KUKA KRL program: EPS_2_25694_HR02_A_20260114065909.src

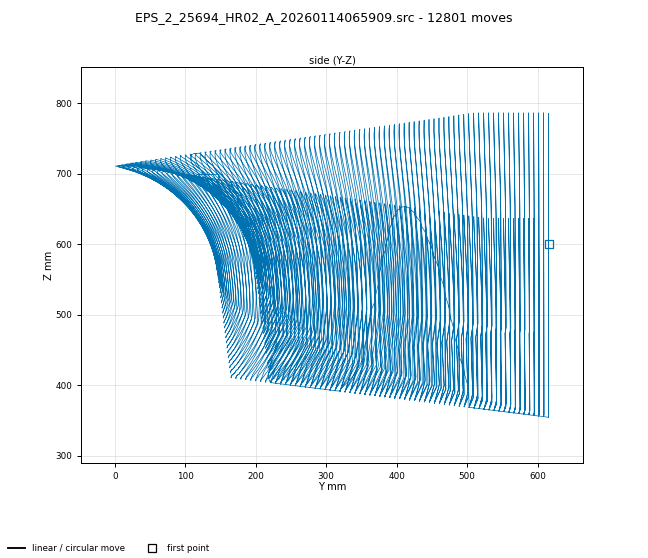
[picture p0: tool path of EPS_2_25694_HR02_A_20260114065909.src, 12801 of 12803 moves have a stored position in this frame; points joined in program order, loops and branches not executed]
&ACCESS RVP
&REL 4
&COMMENT QRS 19112012
&PARAM EDITMASK = *
DEF PART()
EXT BAS (BAS_COMMAND :IN,REAL :IN )
INT I
BAS (#INITMOV,0 )

;KUKA QRS Post kuka4.cps  Date:22-06-2017 !

File_ID=2967

QRS_PRE_INIT()

;Init var - Until changes are made in qrs_pre_init
Outlet_Square_prg=0
Inlet_1_Square_prg=0
Inlet_2_Square_prg=0
Inlet_3_Square_prg=0
Inlet_4_Square_prg=0
Inlet_5_Square_prg=0

Outlet_1={X 0.000, Y 512.360, Z 637.000, B 0.000, E1 0.000 }
Inlet_1={X 0.000, Y 526.980, Z 437.000, B 0.000, E1 171.000 }
Outlet_1_type=299
Inlet_1_type=299
;QRS#1=Sidecore dimensions
;QRS#2=300-12" PVC SDR 35
;QRS#3=300-12" PVC SDR 35
;QRS#4=
;QRS#5=
;QRS#6=
;QRS#7=
;QRS#8=
;QRS#9=16M PSX
;QRS#10=16M PSX
;QRS#11=
;QRS#12=
;QRS#13=
;QRS#14=
;QRS#15=
;QRS#16=1220x127x1067 3,5'
;QRS#17=EPS Height
;QRS#18=786,5
;QRS#19=*
;QRS#20= UPDATED VERSION 22-06-2017
;QRS#21=*
Outlet_Square=0150
Inlet_1_Square=0150
Inlet_2_Square=0
Inlet_3_Square=0
Inlet_4_Square=0
Inlet_5_Square=0
Mill_Square=1
Outlet_Square_Prg=206
Inlet_1_Square_prg=206

QRS_INIT()

$ADVANCE=5

; T1
PTP {E1 173.595,E2 173.595}
PTP {X 0,Y 615.516,A -85,B 0,C 180,E1 173.595,E2 173.595,E3 0,E4 0,E5 0,E6 0}
QRS_SPEED_INIT()
LIN {X 0,Y 615.516,Z 600,A -85,B 0,C 180,E1 173.595,E2 173.595,E3 0,E4 0,E5 0,E6 0} C_VEL
LIN {X 0,Y 615.516,Z 364.494,A -85,B 0,C 180,E1 173.595,E2 173.595} C_VEL
LIN {X 0,Y 615.516,Z 356.327,A -85,B 0,C 180,E1 173.595,E2 173.595} C_VEL
LIN {X 0,Y 615.485,Z 354.327,A -85,B 0,C 180,E1 173.409,E2 173.409} C_VEL
LIN {X 0,Y 615.431,Z 354.324,A -85,B 0,C 180,E1 170.8,E2 170.8} C_VEL
LIN {X 0,Y 615.434,Z 354.324,A -85,B 0,C 180,E1 168.806,E2 168.806} C_VEL
LIN {X 0,Y 615.435,Z 354.324,A -85,B 0,C 180,E1 166.797,E2 166.797} C_VEL
LIN {X 0,Y 615.435,Z 354.324,A -85,B 0,C 180,E1 164.772,E2 164.772} C_VEL
LIN {X 0,Y 615.433,Z 354.323,A -85,B 0,C 180,E1 162.728,E2 162.728} C_VEL
LIN {X 0,Y 615.43,Z 354.323,A -85,B 0,C 180,E1 160.66,E2 160.66} C_VEL
LIN {X 0,Y 615.426,Z 354.323,A -85,B 0,C 180,E1 158.566,E2 158.566} C_VEL
LIN {X 0,Y 615.422,Z 354.322,A -85,B 0,C 180,E1 156.441,E2 156.441} C_VEL
LIN {X 0,Y 615.421,Z 354.322,A -85,B 0,C 180,E1 154.281,E2 154.281} C_VEL
LIN {X 0,Y 615.468,Z 354.319,A -85,B 0,C 180,E1 151.55,E2 151.55} C_VEL
LIN {X 0,Y 615.466,Z 354.324,A -85,B 0,C 180,E1 148.914,E2 148.914} C_VEL
LIN {X 0,Y 615.43,Z 354.322,A -85,B 0,C 180,E1 146.471,E2 146.471} C_VEL
LIN {X 0,Y 615.424,Z 354.321,A -85,B 0,C 180,E1 144.172,E2 144.172} C_VEL
LIN {X 0,Y 615.431,Z 354.32,A -85,B 0,C 180,E1 141.927,E2 141.927} C_VEL
LIN {X 0,Y 615.474,Z 354.319,A -85,B 0,C 180,E1 139.392,E2 139.392} C_VEL
LIN {X 0,Y 615.462,Z 354.324,A -85,B 0,C 180,E1 136.753,E2 136.753} C_VEL
LIN {X 0,Y 615.484,Z 354.326,A -85,B 0,C 180,E1 134.931,E2 134.931} C_VEL
LIN {X 0,Y 615.433,Z 354.322,A -85,B 0,C 180,E1 132.356,E2 132.356} C_VEL
LIN {X 0,Y 615.427,Z 354.32,A -85,B 0,C 180,E1 130.082,E2 130.082} C_VEL
LIN {X 0,Y 615.429,Z 354.32,A -85,B 0,C 180,E1 128.005,E2 128.005} C_VEL
LIN {X 0,Y 615.444,Z 354.318,A -85,B 0,C 180,E1 125.617,E2 125.617} C_VEL
LIN {X 0,Y 615.481,Z 354.318,A -85,B 0,C 180,E1 123.235,E2 123.235} C_VEL
LIN {X 0,Y 615.494,Z 354.325,A -85,B 0,C 180,E1 120.918,E2 120.918} C_VEL
LIN {X 0,Y 615.45,Z 354.322,A -85,B 0,C 180,E1 118.443,E2 118.443} C_VEL
LIN {X 0,Y 615.491,Z 354.505,A -85,B 0,C 180,E1 116.839,E2 116.839} C_VEL
LIN {X 0,Y 615.483,Z 491.228,A -85,B 0,C 180,E1 115.186,E2 115.186} C_VEL
LIN {X 0,Y 615.499,Z 506.898,A -85,B 0,C 180,E1 114.855,E2 114.855} C_VEL
LIN {X 0,Y 615.488,Z 521.69,A -85,B 0,C 180,E1 114.406,E2 114.406} C_VEL
LIN {X 0,Y 615.489,Z 537.106,A -85,B 0,C 180,E1 113.782,E2 113.782} C_VEL
LIN {X 0,Y 615.497,Z 550.263,A -85,B 0,C 180,E1 113.11,E2 113.11} C_VEL
LIN {X 0,Y 615.497,Z 564.134,A -85,B 0,C 180,E1 112.241,E2 112.241} C_VEL
LIN {X 0,Y 615.498,Z 575.987,A -85,B 0,C 180,E1 111.343,E2 111.343} C_VEL
LIN {X 0,Y 615.496,Z 587.548,A -85,B 0,C 180,E1 110.295,E2 110.295} C_VEL
LIN {X 0,Y 615.497,Z 597.952,A -85,B 0,C 180,E1 109.164,E2 109.164} C_VEL
LIN {X 0,Y 615.497,Z 607.204,A -85,B 0,C 180,E1 107.956,E2 107.956} C_VEL
LIN {X 0,Y 615.493,Z 613.803,A -85,B 0,C 180,E1 106.927,E2 106.927} C_VEL
LIN {X 0,Y 615.496,Z 619.357,A -85,B 0,C 180,E1 105.904,E2 105.904} C_VEL
LIN {X 0,Y 615.493,Z 625.35,A -85,B 0,C 180,E1 104.548,E2 104.548} C_VEL
LIN {X 0,Y 615.493,Z 629.892,A -85,B 0,C 180,E1 103.2,E2 103.2} C_VEL
LIN {X 0,Y 615.49,Z 633.115,A -85,B 0,C 180,E1 101.86,E2 101.86} C_VEL
LIN {X 0,Y 615.489,Z 635.059,A -85,B 0,C 180,E1 100.526,E2 100.526} C_VEL
LIN {X 0,Y 615.49,Z 635.837,A -85,B 0,C 180,E1 99.198,E2 99.198} C_VEL
LIN {X 0,Y 615.497,Z 635.466,A -85,B 0,C 180,E1 97.875,E2 97.875} C_VEL
LIN {X 0,Y 615.495,Z 633.965,A -85,B 0,C 180,E1 96.556,E2 96.556} C_VEL
LIN {X 0,Y 615.495,Z 631.316,A -85,B 0,C 180,E1 95.241,E2 95.241} C_VEL
LIN {X 0,Y 615.491,Z 627.446,A -85,B 0,C 180,E1 93.928,E2 93.928} C_VEL
LIN {X 0,Y 615.488,Z 622.26,A -85,B 0,C 180,E1 92.618,E2 92.618} C_VEL
LIN {X 0,Y 615.49,Z 615.673,A -85,B 0,C 180,E1 91.308,E2 91.308} C_VEL
LIN {X 0,Y 615.497,Z 608.611,A -85,B 0,C 180,E1 90.163,E2 90.163} C_VEL
LIN {X 0,Y 615.494,Z 600.168,A -85,B 0,C 180,E1 89.018,E2 89.018} C_VEL
LIN {X 0,Y 615.495,Z 590.053,A -85,B 0,C 180,E1 87.873,E2 87.873} C_VEL
LIN {X 0,Y 615.497,Z 579.74,A -85,B 0,C 180,E1 86.891,E2 86.891} C_VEL
LIN {X 0,Y 615.499,Z 567.432,A -85,B 0,C 180,E1 85.907,E2 85.907} C_VEL
LIN {X 0,Y 615.498,Z 555.113,A -85,B 0,C 180,E1 85.087,E2 85.087} C_VEL
LIN {X 0,Y 615.482,Z 541.656,A -85,B 0,C 180,E1 84.348,E2 84.348} C_VEL
LIN {X 0,Y 615.485,Z 527.73,A -85,B 0,C 180,E1 83.731,E2 83.731} C_VEL
LIN {X 0,Y 615.49,Z 513.077,A -85,B 0,C 180,E1 83.228,E2 83.228} C_VEL
LIN {X 0,Y 615.481,Z 497.717,A -85,B 0,C 180,E1 82.845,E2 82.845} C_VEL
LIN {X 0,Y 615.449,Z 482.279,A -85,B 0,C 180,E1 82.598,E2 82.598} C_VEL
LIN {X 0,Y 615.499,Z 354.424,A -85,B 0,C 180,E1 81.071,E2 81.071} C_VEL
LIN {X 0,Y 615.479,Z 354.321,A -85,B 0,C 180,E1 78.807,E2 78.807} C_VEL
LIN {X 0,Y 615.417,Z 354.323,A -85,B 0,C 180,E1 76.095,E2 76.095} C_VEL
LIN {X 0,Y 615.417,Z 354.323,A -85,B 0,C 180,E1 74.093,E2 74.093} C_VEL
LIN {X 0,Y 615.416,Z 354.323,A -85,B 0,C 180,E1 72.041,E2 72.041} C_VEL
LIN {X 0,Y 615.436,Z 354.324,A -85,B 0,C 180,E1 69.457,E2 69.457} C_VEL
LIN {X 0,Y 615.441,Z 354.322,A -85,B 0,C 180,E1 66.442,E2 66.442} C_VEL
LIN {X 0,Y 615.428,Z 354.323,A -85,B 0,C 180,E1 64.282,E2 64.282} C_VEL
LIN {X 0,Y 615.417,Z 354.323,A -85,B 0,C 180,E1 62.082,E2 62.082} C_VEL
LIN {X 0,Y 615.413,Z 354.323,A -85,B 0,C 180,E1 59.836,E2 59.836} C_VEL
LIN {X 0,Y 615.422,Z 354.324,A -85,B 0,C 180,E1 57.539,E2 57.539} C_VEL
LIN {X 0,Y 615.453,Z 354.325,A -85,B 0,C 180,E1 55.183,E2 55.183} C_VEL
LIN {X 0,Y 615.488,Z 354.324,A -85,B 0,C 180,E1 52.759,E2 52.759} C_VEL
LIN {X 0,Y 615.43,Z 354.323,A -85,B 0,C 180,E1 50.246,E2 50.246} C_VEL
LIN {X 0,Y 615.413,Z 354.324,A -85,B 0,C 180,E1 47.928,E2 47.928} C_VEL
LIN {X 0,Y 615.41,Z 354.324,A -85,B 0,C 180,E1 45.845,E2 45.845} C_VEL
LIN {X 0,Y 615.435,Z 354.325,A -85,B 0,C 180,E1 43.25,E2 43.25} C_VEL
LIN {X 0,Y 615.467,Z 354.326,A -85,B 0,C 180,E1 40.608,E2 40.608} C_VEL
LIN {X 0,Y 615.417,Z 354.324,A -85,B 0,C 180,E1 38.005,E2 38.005} C_VEL
LIN {X 0,Y 615.41,Z 354.324,A -85,B 0,C 180,E1 35.621,E2 35.621} C_VEL
LIN {X 0,Y 615.429,Z 354.325,A -85,B 0,C 180,E1 33.24,E2 33.24} C_VEL
LIN {X 0,Y 615.46,Z 354.326,A -85,B 0,C 180,E1 30.922,E2 30.922} C_VEL
LIN {X 0,Y 615.464,Z 354.325,A -85,B 0,C 180,E1 28.448,E2 28.448} C_VEL
LIN {X 0,Y 615.408,Z 354.325,A -85,B 0,C 180,E1 25.72,E2 25.72} C_VEL
LIN {X 0,Y 615.408,Z 354.325,A -85,B 0,C 180,E1 23.56,E2 23.56} C_VEL
LIN {X 0,Y 615.41,Z 354.325,A -85,B 0,C 180,E1 21.435,E2 21.435} C_VEL
LIN {X 0,Y 615.48,Z 354.328,A -85,B 0,C 180,E1 18.646,E2 18.646} C_VEL
LIN {X 0,Y 615.416,Z 354.325,A -85,B 0,C 180,E1 15.907,E2 15.907} C_VEL
LIN {X 0,Y 615.415,Z 354.325,A -85,B 0,C 180,E1 13.876,E2 13.876} C_VEL
LIN {X 0,Y 615.415,Z 354.325,A -85,B 0,C 180,E1 11.862,E2 11.862} C_VEL
LIN {X 0,Y 615.417,Z 354.325,A -85,B 0,C 180,E1 9.864,E2 9.864} C_VEL
LIN {X 0,Y 615.419,Z 354.325,A -85,B 0,C 180,E1 7.877,E2 7.877} C_VEL
LIN {X 0,Y 615.421,Z 354.325,A -85,B 0,C 180,E1 5.899,E2 5.899} C_VEL
LIN {X 0,Y 615.425,Z 354.325,A -85,B 0,C 180,E1 3.929,E2 3.929} C_VEL
LIN {X 0,Y 615.429,Z 354.325,A -85,B 0,C 180,E1 1.963,E2 1.963} C_VEL
LIN {X 0,Y 615.434,Z 354.325,A -85,B 0,C 180,E1 0,E2 0} C_VEL
LIN {X 0,Y 615.44,Z 354.325,A -85,B 0,C 180,E1 -1.963,E2 -1.963} C_VEL
LIN {X 0,Y 615.41,Z 354.324,A -85,B 0,C 180,E1 -4.585,E2 -4.585} C_VEL
LIN {X 0,Y 615.451,Z 354.323,A -85,B 0,C 180,E1 -7.216,E2 -7.216} C_VEL
LIN {X 0,Y 615.459,Z 354.325,A -85,B 0,C 180,E1 -9.862,E2 -9.862} C_VEL
LIN {X 0,Y 615.411,Z 354.324,A -85,B 0,C 180,E1 -12.532,E2 -12.532} C_VEL
LIN {X 0,Y 615.412,Z 354.324,A -85,B 0,C 180,E1 -14.551,E2 -14.551} C_VEL
LIN {X 0,Y 615.411,Z 354.324,A -85,B 0,C 180,E1 -16.589,E2 -16.589} C_VEL
LIN {X 0,Y 615.458,Z 354.323,A -85,B 0,C 180,E1 -19.339,E2 -19.339} C_VEL
LIN {X 0,Y 615.438,Z 354.324,A -85,B 0,C 180,E1 -22.138,E2 -22.138} C_VEL
LIN {X 0,Y 615.428,Z 354.324,A -85,B 0,C 180,E1 -24.274,E2 -24.274} C_VEL
LIN {X 0,Y 615.418,Z 354.324,A -85,B 0,C 180,E1 -26.447,E2 -26.447} C_VEL
LIN {X 0,Y 615.414,Z 354.323,A -85,B 0,C 180,E1 -28.662,E2 -28.662} C_VEL
LIN {X 0,Y 615.418,Z 354.323,A -85,B 0,C 180,E1 -30.923,E2 -30.923} C_VEL
LIN {X 0,Y 615.471,Z 354.322,A -85,B 0,C 180,E1 -33.534,E2 -33.534} C_VEL
LIN {X 0,Y 615.482,Z 354.328,A -85,B 0,C 180,E1 -35.835,E2 -35.835} C_VEL
LIN {X 0,Y 615.457,Z 354.325,A -85,B 0,C 180,E1 -38.071,E2 -38.071} C_VEL
LIN {X 0,Y 615.46,Z 354.324,A -85,B 0,C 180,E1 -40.087,E2 -40.087} C_VEL
LIN {X 0,Y 615.434,Z 354.324,A -85,B 0,C 180,E1 -42.357,E2 -42.357} C_VEL
LIN {X 0,Y 615.418,Z 354.322,A -85,B 0,C 180,E1 -44.926,E2 -44.926} C_VEL
LIN {X 0,Y 615.418,Z 354.322,A -85,B 0,C 180,E1 -46.959,E2 -46.959} C_VEL
LIN {X 0,Y 615.446,Z 354.321,A -85,B 0,C 180,E1 -49.391,E2 -49.391} C_VEL
LIN {X 0,Y 615.478,Z 354.327,A -85,B 0,C 180,E1 -51.989,E2 -51.989} C_VEL
LIN {X 0,Y 615.44,Z 354.324,A -85,B 0,C 180,E1 -54.382,E2 -54.382} C_VEL
LIN {X 0,Y 615.418,Z 354.323,A -85,B 0,C 180,E1 -56.76,E2 -56.76} C_VEL
LIN {X 0,Y 615.42,Z 354.322,A -85,B 0,C 180,E1 -59.077,E2 -59.077} C_VEL
LIN {X 0,Y 615.42,Z 354.346,A -85,B 0,C 180,E1 -61.012,E2 -61.012} C_VEL
LIN {X 0,Y 615.481,Z 379.996,A -85,B 0,C 180,E1 -63.408,E2 -63.408} C_VEL
LIN {X 0,Y 615.492,Z 410.8,A -85,B 0,C 180,E1 -66.217,E2 -66.217} C_VEL
LIN {X 0,Y 615.498,Z 441.071,A -85,B 0,C 180,E1 -68.92,E2 -68.92} C_VEL
LIN {X 0,Y 615.486,Z 473.336,A -85,B 0,C 180,E1 -71.741,E2 -71.741} C_VEL
LIN {X 0,Y 615.485,Z 641.171,A -85,B 0,C 180,E1 -73.768,E2 -73.768} C_VEL
LIN {X 0,Y 615.487,Z 656.72,A -85,B 0,C 180,E1 -74.095,E2 -74.095} C_VEL
LIN {X 0,Y 615.479,Z 672.055,A -85,B 0,C 180,E1 -74.562,E2 -74.562} C_VEL
LIN {X 0,Y 615.484,Z 685.757,A -85,B 0,C 180,E1 -75.113,E2 -75.113} C_VEL
LIN {X 0,Y 615.493,Z 700.047,A -85,B 0,C 180,E1 -75.834,E2 -75.834} C_VEL
LIN {X 0,Y 615.497,Z 712.9,A -85,B 0,C 180,E1 -76.631,E2 -76.631} C_VEL
LIN {X 0,Y 615.495,Z 725.256,A -85,B 0,C 180,E1 -77.554,E2 -77.554} C_VEL
LIN {X 0,Y 615.495,Z 735.607,A -85,B 0,C 180,E1 -78.473,E2 -78.473} C_VEL
LIN {X 0,Y 615.494,Z 745.184,A -85,B 0,C 180,E1 -79.473,E2 -79.473} C_VEL
LIN {X 0,Y 615.495,Z 754.577,A -85,B 0,C 180,E1 -80.636,E2 -80.636} C_VEL
LIN {X 0,Y 615.495,Z 762.38,A -85,B 0,C 180,E1 -81.794,E2 -81.794} C_VEL
LIN {X 0,Y 615.497,Z 769.607,A -85,B 0,C 180,E1 -83.102,E2 -83.102} C_VEL
LIN {X 0,Y 615.499,Z 775.436,A -85,B 0,C 180,E1 -84.43,E2 -84.43} C_VEL
LIN {X 0,Y 615.491,Z 778.86,A -85,B 0,C 180,E1 -85.415,E2 -85.415} C_VEL
LIN {X 0,Y 615.492,Z 782.318,A -85,B 0,C 180,E1 -86.727,E2 -86.727} C_VEL
LIN {X 0,Y 615.495,Z 784.593,A -85,B 0,C 180,E1 -88.037,E2 -88.037} C_VEL
LIN {X 0,Y 615.493,Z 785.74,A -85,B 0,C 180,E1 -89.346,E2 -89.346} C_VEL
LIN {X 0,Y 615.493,Z 785.741,A -85,B 0,C 180,E1 -90.654,E2 -90.654} C_VEL
LIN {X 0,Y 615.495,Z 784.594,A -85,B 0,C 180,E1 -91.963,E2 -91.963} C_VEL
LIN {X 0,Y 615.492,Z 782.319,A -85,B 0,C 180,E1 -93.273,E2 -93.273} C_VEL
LIN {X 0,Y 615.491,Z 778.861,A -85,B 0,C 180,E1 -94.584,E2 -94.584} C_VEL
LIN {X 0,Y 615.49,Z 774.145,A -85,B 0,C 180,E1 -95.898,E2 -95.898} C_VEL
LIN {X 0,Y 615.496,Z 768.031,A -85,B 0,C 180,E1 -97.215,E2 -97.215} C_VEL
LIN {X 0,Y 615.49,Z 760.336,A -85,B 0,C 180,E1 -98.536,E2 -98.536} C_VEL
LIN {X 0,Y 615.495,Z 752.117,A -85,B 0,C 180,E1 -99.696,E2 -99.696} C_VEL
LIN {X 0,Y 615.496,Z 741.897,A -85,B 0,C 180,E1 -100.892,E2 -100.892} C_VEL
LIN {X 0,Y 615.495,Z 732.073,A -85,B 0,C 180,E1 -101.86,E2 -101.86} C_VEL
LIN {X 0,Y 615.497,Z 719.955,A -85,B 0,C 180,E1 -102.865,E2 -102.865} C_VEL
LIN {X 0,Y 615.498,Z 707.807,A -85,B 0,C 180,E1 -103.705,E2 -103.705} C_VEL
LIN {X 0,Y 615.477,Z 694.39,A -85,B 0,C 180,E1 -104.472,E2 -104.472} C_VEL
LIN {X 0,Y 615.495,Z 679.863,A -85,B 0,C 180,E1 -105.14,E2 -105.14} C_VEL
LIN {X 0,Y 615.477,Z 665.636,A -85,B 0,C 180,E1 -105.65,E2 -105.65} C_VEL
LIN {X 0,Y 615.495,Z 651.162,A -85,B 0,C 180,E1 -106.035,E2 -106.035} C_VEL
LIN {X 0,Y 615.485,Z 636.614,A -85,B 0,C 180,E1 -106.297,E2 -106.297} C_VEL
LIN {X 0,Y 615.486,Z 473.045,A -85,B 0,C 180,E1 -108.279,E2 -108.279} C_VEL
LIN {X 0,Y 615.498,Z 441.077,A -85,B 0,C 180,E1 -111.08,E2 -111.08} C_VEL
LIN {X 0,Y 615.495,Z 408.281,A -85,B 0,C 180,E1 -114.01,E2 -114.01} C_VEL
LIN {X 0,Y 615.474,Z 378.393,A -85,B 0,C 180,E1 -116.74,E2 -116.74} C_VEL
LIN {X 0,Y 615.419,Z 354.322,A -85,B 0,C 180,E1 -118.999,E2 -118.999} C_VEL
LIN {X 0,Y 615.417,Z 354.323,A -85,B 0,C 180,E1 -121.075,E2 -121.075} C_VEL
LIN {X 0,Y 615.433,Z 354.324,A -85,B 0,C 180,E1 -123.527,E2 -123.527} C_VEL
LIN {X 0,Y 615.466,Z 354.321,A -85,B 0,C 180,E1 -126.425,E2 -126.425} C_VEL
LIN {X 0,Y 615.422,Z 354.322,A -85,B 0,C 180,E1 -128.908,E2 -128.908} C_VEL
LIN {X 0,Y 615.416,Z 354.323,A -85,B 0,C 180,E1 -131.087,E2 -131.087} C_VEL
LIN {X 0,Y 615.414,Z 354.323,A -85,B 0,C 180,E1 -133.249,E2 -133.249} C_VEL
LIN {X 0,Y 615.415,Z 354.323,A -85,B 0,C 180,E1 -135.073,E2 -135.073} C_VEL
LIN {X 0,Y 615.429,Z 354.324,A -85,B 0,C 180,E1 -137.642,E2 -137.642} C_VEL
LIN {X 0,Y 615.496,Z 354.324,A -85,B 0,C 180,E1 -140.251,E2 -140.251} C_VEL
LIN {X 0,Y 615.415,Z 354.324,A -85,B 0,C 180,E1 -143.07,E2 -143.07} C_VEL
LIN {X 0,Y 615.408,Z 354.325,A -85,B 0,C 180,E1 -145.308,E2 -145.308} C_VEL
LIN {X 0,Y 615.422,Z 354.325,A -85,B 0,C 180,E1 -147.676,E2 -147.676} C_VEL
LIN {X 0,Y 615.459,Z 354.324,A -85,B 0,C 180,E1 -150.592,E2 -150.592} C_VEL
LIN {X 0,Y 615.421,Z 354.324,A -85,B 0,C 180,E1 -152.964,E2 -152.964} C_VEL
LIN {X 0,Y 615.419,Z 354.325,A -85,B 0,C 180,E1 -155.005,E2 -155.005} C_VEL
LIN {X 0,Y 615.411,Z 354.325,A -85,B 0,C 180,E1 -157.153,E2 -157.153} C_VEL
LIN {X 0,Y 615.407,Z 354.325,A -85,B 0,C 180,E1 -159.459,E2 -159.459} C_VEL
LIN {X 0,Y 615.445,Z 354.325,A -85,B 0,C 180,E1 -162.042,E2 -162.042} C_VEL
LIN {X 0,Y 615.448,Z 354.325,A -85,B 0,C 180,E1 -164.773,E2 -164.773} C_VEL
LIN {X 0,Y 615.409,Z 354.324,A -85,B 0,C 180,E1 -167.468,E2 -167.468} C_VEL
LIN {X 0,Y 615.449,Z 354.324,A -85,B 0,C 180,E1 -170.137,E2 -170.137} C_VEL
LIN {X 0,Y 615.457,Z 354.325,A -85,B 0,C 180,E1 -172.784,E2 -172.784} C_VEL
LIN {X 0,Y 615.412,Z 354.324,A -85,B 0,C 180,E1 -175.415,E2 -175.415} C_VEL
LIN {X 0,Y 615.412,Z 354.324,A -85,B 0,C 180,E1 -177.382,E2 -177.382} C_VEL
LIN {X 0,Y 615.416,Z 354.324,A -85,B 0,C 180,E1 -179.346,E2 -179.346} C_VEL
LIN {X 0,Y 615.419,Z 354.324,A -85,B 0,C 180,E1 -181.309,E2 -181.309} C_VEL
LIN {X 0,Y 615.422,Z 354.324,A -85,B 0,C 180,E1 -183.273,E2 -183.273} C_VEL
LIN {X 0,Y 615.425,Z 354.324,A -85,B 0,C 180,E1 -185.242,E2 -185.242} C_VEL
LIN {X 0,Y 615.485,Z 354.327,A -85,B 0,C 180,E1 -186.591,E2 -186.591} C_VEL
LIN {X 0,Y 614.772,Z 354.467,A -85,B 0,C 180,E1 -187.137,E2 -187.137} C_VEL
LIN {X 0,Y 611.914,Z 354.882,A -85,B 0,C 180,E1 -188.023,E2 -188.023} C_VEL
LIN {X 0,Y 609.525,Z 355.191,A -85,B 0,C 180,E1 -188.735,E2 -188.735} C_VEL
LIN {X 0,Y 608.494,Z 355.309,A -85,B 0,C 180,E1 -189.285,E2 -189.285} C_VEL
LIN {X 0,Y 608.406,Z 355.318,A -85,B 0,C 180,E1 -189.471,E2 -189.471} C_VEL
LIN {X 0,Y 608.416,Z 355.317,A -85,B 0,C 180,E1 -192.001,E2 -192.001} C_VEL
LIN {X 0,Y 608.458,Z 355.322,A -85,B 0,C 180,E1 -194.721,E2 -194.721} C_VEL
LIN {X 0,Y 608.402,Z 355.319,A -85,B 0,C 180,E1 -197.478,E2 -197.478} C_VEL
LIN {X 0,Y 608.4,Z 355.318,A -85,B 0,C 180,E1 -199.573,E2 -199.573} C_VEL
LIN {X 0,Y 608.417,Z 355.316,A -85,B 0,C 180,E1 -201.694,E2 -201.694} C_VEL
LIN {X 0,Y 608.429,Z 355.322,A -85,B 0,C 180,E1 -204.572,E2 -204.572} C_VEL
LIN {X 0,Y 608.409,Z 355.318,A -85,B 0,C 180,E1 -207.52,E2 -207.52} C_VEL
LIN {X 0,Y 608.412,Z 355.317,A -85,B 0,C 180,E1 -209.966,E2 -209.966} C_VEL
LIN {X 0,Y 608.443,Z 355.318,A -85,B 0,C 180,E1 -212.522,E2 -212.522} C_VEL
LIN {X 0,Y 608.414,Z 355.321,A -85,B 0,C 180,E1 -215.28,E2 -215.28} C_VEL
LIN {X 0,Y 608.424,Z 355.316,A -85,B 0,C 180,E1 -217.75,E2 -217.75} C_VEL
LIN {X 0,Y 608.423,Z 355.317,A -85,B 0,C 180,E1 -220.328,E2 -220.328} C_VEL
LIN {X 0,Y 608.45,Z 355.317,A -85,B 0,C 180,E1 -223.309,E2 -223.309} C_VEL
LIN {X 0,Y 608.405,Z 355.318,A -85,B 0,C 180,E1 -225.741,E2 -225.741} C_VEL
LIN {X 0,Y 608.411,Z 355.317,A -85,B 0,C 180,E1 -227.936,E2 -227.936} C_VEL
LIN {X 0,Y 608.439,Z 355.319,A -85,B 0,C 180,E1 -230.707,E2 -230.707} C_VEL
LIN {X 0,Y 608.454,Z 355.323,A -85,B 0,C 180,E1 -233.086,E2 -233.086} C_VEL
LIN {X 0,Y 608.443,Z 355.317,A -85,B 0,C 180,E1 -235.53,E2 -235.53} C_VEL
LIN {X 0,Y 608.424,Z 355.316,A -85,B 0,C 180,E1 -237.904,E2 -237.904} C_VEL
LIN {X 0,Y 608.423,Z 355.316,A -85,B 0,C 180,E1 -240.219,E2 -240.219} C_VEL
LIN {X 0,Y 608.468,Z 355.318,A -85,B 0,C 180,E1 -242.941,E2 -242.941} C_VEL
LIN {X 0,Y 608.741,Z 357.487,A -85,B 0,C 180,E1 -242.992,E2 -242.992} C_VEL
LIN {X 0,Y 608.678,Z 490.791,A -85,B 0,C 180,E1 -244.62,E2 -244.62} C_VEL
LIN {X 0,Y 608.659,Z 506.862,A -85,B 0,C 180,E1 -244.961,E2 -244.961} C_VEL
LIN {X 0,Y 608.626,Z 522.288,A -85,B 0,C 180,E1 -245.437,E2 -245.437} C_VEL
LIN {X 0,Y 608.585,Z 537.11,A -85,B 0,C 180,E1 -246.046,E2 -246.046} C_VEL
LIN {X 0,Y 608.57,Z 551.423,A -85,B 0,C 180,E1 -246.792,E2 -246.792} C_VEL
LIN {X 0,Y 608.56,Z 564.104,A -85,B 0,C 180,E1 -247.599,E2 -247.599} C_VEL
LIN {X 0,Y 608.518,Z 576.847,A -85,B 0,C 180,E1 -248.578,E2 -248.578} C_VEL
LIN {X 0,Y 608.496,Z 587.915,A -85,B 0,C 180,E1 -249.595,E2 -249.595} C_VEL
LIN {X 0,Y 608.485,Z 597.257,A -85,B 0,C 180,E1 -250.607,E2 -250.607} C_VEL
LIN {X 0,Y 608.465,Z 606.755,A -85,B 0,C 180,E1 -251.829,E2 -251.829} C_VEL
LIN {X 0,Y 608.458,Z 614.547,A -85,B 0,C 180,E1 -253.044,E2 -253.044} C_VEL
LIN {X 0,Y 608.432,Z 620.919,A -85,B 0,C 180,E1 -254.25,E2 -254.25} C_VEL
LIN {X 0,Y 608.428,Z 626.707,A -85,B 0,C 180,E1 -255.621,E2 -255.621} C_VEL
LIN {X 0,Y 608.44,Z 630.134,A -85,B 0,C 180,E1 -256.644,E2 -256.644} C_VEL
LIN {X 0,Y 608.435,Z 633.461,A -85,B 0,C 180,E1 -258,E2 -258} C_VEL
LIN {X 0,Y 608.432,Z 635.534,A -85,B 0,C 180,E1 -259.35,E2 -259.35} C_VEL
LIN {X 0,Y 608.413,Z 636.424,A -85,B 0,C 180,E1 -260.694,E2 -260.694} C_VEL
LIN {X 0,Y 608.42,Z 636.149,A -85,B 0,C 180,E1 -262.033,E2 -262.033} C_VEL
LIN {X 0,Y 608.446,Z 634.676,A -85,B 0,C 180,E1 -263.398,E2 -263.398} C_VEL
LIN {X 0,Y 608.437,Z 632.138,A -85,B 0,C 180,E1 -264.698,E2 -264.698} C_VEL
LIN {X 0,Y 608.43,Z 628.287,A -85,B 0,C 180,E1 -266.026,E2 -266.026} C_VEL
LIN {X 0,Y 608.424,Z 623.155,A -85,B 0,C 180,E1 -267.352,E2 -267.352} C_VEL
LIN {X 0,Y 608.444,Z 616.62,A -85,B 0,C 180,E1 -268.677,E2 -268.677} C_VEL
LIN {X 0,Y 608.465,Z 608.515,A -85,B 0,C 180,E1 -270,E2 -270} C_VEL
LIN {X 0,Y 608.476,Z 599.915,A -85,B 0,C 180,E1 -271.158,E2 -271.158} C_VEL
LIN {X 0,Y 608.482,Z 589.638,A -85,B 0,C 180,E1 -272.317,E2 -272.317} C_VEL
LIN {X 0,Y 608.518,Z 579.153,A -85,B 0,C 180,E1 -273.311,E2 -273.311} C_VEL
LIN {X 0,Y 608.549,Z 566.658,A -85,B 0,C 180,E1 -274.305,E2 -274.305} C_VEL
LIN {X 0,Y 608.558,Z 554.13,A -85,B 0,C 180,E1 -275.135,E2 -275.135} C_VEL
LIN {X 0,Y 608.587,Z 540.409,A -85,B 0,C 180,E1 -275.883,E2 -275.883} C_VEL
LIN {X 0,Y 608.62,Z 526.427,A -85,B 0,C 180,E1 -276.495,E2 -276.495} C_VEL
LIN {X 0,Y 608.652,Z 511.473,A -85,B 0,C 180,E1 -276.999,E2 -276.999} C_VEL
LIN {X 0,Y 608.651,Z 496.73,A -85,B 0,C 180,E1 -277.36,E2 -277.36} C_VEL
LIN {X 0,Y 608.645,Z 480.598,A -85,B 0,C 180,E1 -277.61,E2 -277.61} C_VEL
LIN {X 0,Y 608.664,Z 356.307,A -85,B 0,C 180,E1 -279.114,E2 -279.114} C_VEL
LIN {X 0,Y 608.453,Z 355.32,A -85,B 0,C 180,E1 -279.138,E2 -279.138} C_VEL
LIN {X 0,Y 608.434,Z 355.319,A -85,B 0,C 180,E1 -281.325,E2 -281.325} C_VEL
LIN {X 0,Y 608.391,Z 355.32,A -85,B 0,C 180,E1 -284.039,E2 -284.039} C_VEL
LIN {X 0,Y 608.434,Z 355.318,A -85,B 0,C 180,E1 -286.517,E2 -286.517} C_VEL
LIN {X 0,Y 608.417,Z 355.319,A -85,B 0,C 180,E1 -289.572,E2 -289.572} C_VEL
LIN {X 0,Y 608.425,Z 355.317,A -85,B 0,C 180,E1 -291.693,E2 -291.693} C_VEL
LIN {X 0,Y 608.422,Z 355.319,A -85,B 0,C 180,E1 -294.572,E2 -294.572} C_VEL
LIN {X 0,Y 608.422,Z 355.319,A -85,B 0,C 180,E1 -297.519,E2 -297.519} C_VEL
LIN {X 0,Y 608.391,Z 355.319,A -85,B 0,C 180,E1 -299.958,E2 -299.958} C_VEL
LIN {X 0,Y 608.408,Z 355.319,A -85,B 0,C 180,E1 -302.514,E2 -302.514} C_VEL
LIN {X 0,Y 608.408,Z 355.326,A -85,B 0,C 180,E1 -305.279,E2 -305.279} C_VEL
LIN {X 0,Y 608.425,Z 355.317,A -85,B 0,C 180,E1 -307.749,E2 -307.749} C_VEL
LIN {X 0,Y 608.398,Z 355.319,A -85,B 0,C 180,E1 -310.323,E2 -310.323} C_VEL
LIN {X 0,Y 608.43,Z 355.322,A -85,B 0,C 180,E1 -312.961,E2 -312.961} C_VEL
LIN {X 0,Y 608.405,Z 355.32,A -85,B 0,C 180,E1 -315.74,E2 -315.74} C_VEL
LIN {X 0,Y 608.405,Z 355.319,A -85,B 0,C 180,E1 -317.934,E2 -317.934} C_VEL
LIN {X 0,Y 608.408,Z 355.32,A -85,B 0,C 180,E1 -320.708,E2 -320.708} C_VEL
LIN {X 0,Y 608.432,Z 355.322,A -85,B 0,C 180,E1 -323.083,E2 -323.083} C_VEL
LIN {X 0,Y 608.448,Z 355.319,A -85,B 0,C 180,E1 -325.529,E2 -325.529} C_VEL
LIN {X 0,Y 608.417,Z 355.318,A -85,B 0,C 180,E1 -327.902,E2 -327.902} C_VEL
LIN {X 0,Y 608.397,Z 355.319,A -85,B 0,C 180,E1 -330.216,E2 -330.216} C_VEL
LIN {X 0,Y 608.396,Z 355.319,A -85,B 0,C 180,E1 -332.479,E2 -332.479} C_VEL
LIN {X 0,Y 608.418,Z 355.326,A -85,B 0,C 180,E1 -335.427,E2 -335.427} C_VEL
LIN {X 0,Y 608.406,Z 355.318,A -85,B 0,C 180,E1 -338.306,E2 -338.306} C_VEL
LIN {X 0,Y 608.388,Z 355.32,A -85,B 0,C 180,E1 -340.427,E2 -340.427} C_VEL
LIN {X 0,Y 608.389,Z 355.32,A -85,B 0,C 180,E1 -342.521,E2 -342.521} C_VEL
LIN {X 0,Y 608.407,Z 355.318,A -85,B 0,C 180,E1 -344.592,E2 -344.592} C_VEL
LIN {X 0,Y 608.458,Z 355.32,A -85,B 0,C 180,E1 -347.322,E2 -347.322} C_VEL
LIN {X 0,Y 608.401,Z 355.32,A -85,B 0,C 180,E1 -350.022,E2 -350.022} C_VEL
LIN {X 0,Y 608.393,Z 355.321,A -85,B 0,C 180,E1 -352.032,E2 -352.032} C_VEL
LIN {X 0,Y 608.404,Z 355.32,A -85,B 0,C 180,E1 -354.032,E2 -354.032} C_VEL
LIN {X 0,Y 608.398,Z 355.321,A -85,B 0,C 180,E1 -356.025,E2 -356.025} C_VEL
LIN {X 0,Y 608.403,Z 355.321,A -85,B 0,C 180,E1 -358.014,E2 -358.014} C_VEL
LIN {X 0,Y 608.429,Z 355.318,A -85,B 0,C 180,E1 -360,E2 -360} C_VEL
LIN {X 0,Y 608.409,Z 355.317,A -85,B 0,C 180,E1 -362.648,E2 -362.648} C_VEL
LIN {X 0,Y 608.435,Z 355.32,A -85,B 0,C 180,E1 -365.302,E2 -365.302} C_VEL
LIN {X 0,Y 608.415,Z 355.321,A -85,B 0,C 180,E1 -367.968,E2 -367.968} C_VEL
LIN {X 0,Y 608.395,Z 355.319,A -85,B 0,C 180,E1 -370.651,E2 -370.651} C_VEL
LIN {X 0,Y 608.428,Z 355.321,A -85,B 0,C 180,E1 -373.357,E2 -373.357} C_VEL
LIN {X 0,Y 608.419,Z 355.32,A -85,B 0,C 180,E1 -376.095,E2 -376.095} C_VEL
LIN {X 0,Y 608.415,Z 355.317,A -85,B 0,C 180,E1 -378.871,E2 -378.871} C_VEL
LIN {X 0,Y 608.442,Z 355.325,A -85,B 0,C 180,E1 -381.692,E2 -381.692} C_VEL
LIN {X 0,Y 608.401,Z 355.319,A -85,B 0,C 180,E1 -384.573,E2 -384.573} C_VEL
LIN {X 0,Y 608.385,Z 355.32,A -85,B 0,C 180,E1 -386.777,E2 -386.777} C_VEL
LIN {X 0,Y 608.473,Z 355.32,A -85,B 0,C 180,E1 -389.779,E2 -389.779} C_VEL
LIN {X 0,Y 608.404,Z 355.319,A -85,B 0,C 180,E1 -392.516,E2 -392.516} C_VEL
LIN {X 0,Y 608.388,Z 355.32,A -85,B 0,C 180,E1 -394.899,E2 -394.899} C_VEL
LIN {X 0,Y 608.426,Z 355.317,A -85,B 0,C 180,E1 -397.154,E2 -397.154} C_VEL
LIN {X 0,Y 608.425,Z 355.318,A -85,B 0,C 180,E1 -400.327,E2 -400.327} C_VEL
LIN {X 0,Y 608.389,Z 355.32,A -85,B 0,C 180,E1 -402.965,E2 -402.965} C_VEL
LIN {X 0,Y 608.458,Z 355.32,A -85,B 0,C 180,E1 -405.736,E2 -405.736} C_VEL
LIN {X 0,Y 608.472,Z 355.32,A -85,B 0,C 180,E1 -407.941,E2 -407.941} C_VEL
LIN {X 0,Y 608.398,Z 355.319,A -85,B 0,C 180,E1 -410.711,E2 -410.711} C_VEL
LIN {X 0,Y 608.394,Z 355.32,A -85,B 0,C 180,E1 -413.081,E2 -413.081} C_VEL
LIN {X 0,Y 608.439,Z 355.318,A -85,B 0,C 180,E1 -415.529,E2 -415.529} C_VEL
LIN {X 0,Y 608.45,Z 355.323,A -85,B 0,C 180,E1 -417.905,E2 -417.905} C_VEL
LIN {X 0,Y 608.395,Z 355.337,A -85,B 0,C 180,E1 -420.74,E2 -420.74} C_VEL
LIN {X 0,Y 608.818,Z 359.499,A -85,B 0,C 180,E1 -421.159,E2 -421.159} C_VEL
LIN {X 0,Y 608.798,Z 387.549,A -85,B 0,C 180,E1 -423.797,E2 -423.797} C_VEL
LIN {X 0,Y 608.74,Z 417.283,A -85,B 0,C 180,E1 -426.528,E2 -426.528} C_VEL
LIN {X 0,Y 608.657,Z 449.974,A -85,B 0,C 180,E1 -429.467,E2 -429.467} C_VEL
LIN {X 0,Y 608.601,Z 473.336,A -85,B 0,C 180,E1 -431.527,E2 -431.527} C_VEL
LIN {X 0,Y 608.682,Z 621.009,A -85,B 0,C 180,E1 -433.32,E2 -433.32} C_VEL
LIN {X 0,Y 608.672,Z 642.946,A -85,B 0,C 180,E1 -433.614,E2 -433.614} C_VEL
LIN {X 0,Y 608.639,Z 658.255,A -85,B 0,C 180,E1 -433.954,E2 -433.954} C_VEL
LIN {X 0,Y 608.604,Z 673.188,A -85,B 0,C 180,E1 -434.426,E2 -434.426} C_VEL
LIN {X 0,Y 608.588,Z 687.617,A -85,B 0,C 180,E1 -435.026,E2 -435.026} C_VEL
LIN {X 0,Y 608.563,Z 700.792,A -85,B 0,C 180,E1 -435.709,E2 -435.709} C_VEL
LIN {X 0,Y 608.548,Z 714.201,A -85,B 0,C 180,E1 -436.561,E2 -436.561} C_VEL
LIN {X 0,Y 608.504,Z 726.389,A -85,B 0,C 180,E1 -437.493,E2 -437.493} C_VEL
LIN {X 0,Y 608.496,Z 737.51,A -85,B 0,C 180,E1 -438.508,E2 -438.508} C_VEL
LIN {X 0,Y 608.476,Z 748.299,A -85,B 0,C 180,E1 -439.687,E2 -439.687} C_VEL
LIN {X 0,Y 608.47,Z 757.29,A -85,B 0,C 180,E1 -440.862,E2 -440.862} C_VEL
LIN {X 0,Y 608.458,Z 764.752,A -85,B 0,C 180,E1 -442.033,E2 -442.033} C_VEL
LIN {X 0,Y 608.44,Z 771.86,A -85,B 0,C 180,E1 -443.399,E2 -443.399} C_VEL
LIN {X 0,Y 608.437,Z 777.16,A -85,B 0,C 180,E1 -444.698,E2 -444.698} C_VEL
LIN {X 0,Y 608.431,Z 781.287,A -85,B 0,C 180,E1 -446.026,E2 -446.026} C_VEL
LIN {X 0,Y 608.423,Z 784.184,A -85,B 0,C 180,E1 -447.352,E2 -447.352} C_VEL
LIN {X 0,Y 608.445,Z 785.912,A -85,B 0,C 180,E1 -448.676,E2 -448.676} C_VEL
LIN {X 0,Y 608.431,Z 786.5,A -85,B 0,C 180,E1 -450,E2 -450} C_VEL
LIN {X 0,Y 608.445,Z 785.912,A -85,B 0,C 180,E1 -451.323,E2 -451.323} C_VEL
LIN {X 0,Y 608.423,Z 784.185,A -85,B 0,C 180,E1 -452.648,E2 -452.648} C_VEL
LIN {X 0,Y 608.431,Z 781.288,A -85,B 0,C 180,E1 -453.974,E2 -453.974} C_VEL
LIN {X 0,Y 608.437,Z 777.162,A -85,B 0,C 180,E1 -455.302,E2 -455.302} C_VEL
LIN {X 0,Y 608.436,Z 771.705,A -85,B 0,C 180,E1 -456.633,E2 -456.633} C_VEL
LIN {X 0,Y 608.457,Z 764.755,A -85,B 0,C 180,E1 -457.967,E2 -457.967} C_VEL
LIN {X 0,Y 608.47,Z 757.293,A -85,B 0,C 180,E1 -459.138,E2 -459.138} C_VEL
LIN {X 0,Y 608.476,Z 748.303,A -85,B 0,C 180,E1 -460.313,E2 -460.313} C_VEL
LIN {X 0,Y 608.496,Z 737.515,A -85,B 0,C 180,E1 -461.492,E2 -461.492} C_VEL
LIN {X 0,Y 608.504,Z 726.396,A -85,B 0,C 180,E1 -462.506,E2 -462.506} C_VEL
LIN {X 0,Y 608.548,Z 714.209,A -85,B 0,C 180,E1 -463.439,E2 -463.439} C_VEL
LIN {X 0,Y 608.57,Z 701.232,A -85,B 0,C 180,E1 -464.265,E2 -464.265} C_VEL
LIN {X 0,Y 608.588,Z 687.627,A -85,B 0,C 180,E1 -464.974,E2 -464.974} C_VEL
LIN {X 0,Y 608.604,Z 673.202,A -85,B 0,C 180,E1 -465.573,E2 -465.573} C_VEL
LIN {X 0,Y 608.639,Z 658.276,A -85,B 0,C 180,E1 -466.045,E2 -466.045} C_VEL
LIN {X 0,Y 608.672,Z 642.959,A -85,B 0,C 180,E1 -466.385,E2 -466.385} C_VEL
LIN {X 0,Y 608.672,Z 616.719,A -85,B 0,C 180,E1 -466.732,E2 -466.732} C_VEL
LIN {X 0,Y 608.723,Z 474.092,A -85,B 0,C 180,E1 -468.46,E2 -468.46} C_VEL
LIN {X 0,Y 608.584,Z 473.045,A -85,B 0,C 180,E1 -468.493,E2 -468.493} C_VEL
LIN {X 0,Y 608.665,Z 443.059,A -85,B 0,C 180,E1 -471.15,E2 -471.15} C_VEL
LIN {X 0,Y 608.751,Z 410.803,A -85,B 0,C 180,E1 -474.062,E2 -474.062} C_VEL
LIN {X 0,Y 608.804,Z 380.001,A -85,B 0,C 180,E1 -476.907,E2 -476.907} C_VEL
LIN {X 0,Y 608.81,Z 357.821,A -85,B 0,C 180,E1 -479.001,E2 -479.001} C_VEL
LIN {X 0,Y 608.398,Z 355.322,A -85,B 0,C 180,E1 -479.283,E2 -479.283} C_VEL
LIN {X 0,Y 608.419,Z 355.317,A -85,B 0,C 180,E1 -481.318,E2 -481.318} C_VEL
LIN {X 0,Y 608.439,Z 355.319,A -85,B 0,C 180,E1 -483.73,E2 -483.73} C_VEL
LIN {X 0,Y 608.434,Z 355.325,A -85,B 0,C 180,E1 -486.092,E2 -486.092} C_VEL
LIN {X 0,Y 608.402,Z 355.321,A -85,B 0,C 180,E1 -488.592,E2 -488.592} C_VEL
LIN {X 0,Y 608.386,Z 355.32,A -85,B 0,C 180,E1 -491.181,E2 -491.181} C_VEL
LIN {X 0,Y 608.411,Z 355.317,A -85,B 0,C 180,E1 -493.303,E2 -493.303} C_VEL
LIN {X 0,Y 608.449,Z 355.323,A -85,B 0,C 180,E1 -496.129,E2 -496.129} C_VEL
LIN {X 0,Y 608.4,Z 355.32,A -85,B 0,C 180,E1 -498.819,E2 -498.819} C_VEL
LIN {X 0,Y 608.384,Z 355.321,A -85,B 0,C 180,E1 -501.406,E2 -501.406} C_VEL
LIN {X 0,Y 608.429,Z 355.321,A -85,B 0,C 180,E1 -503.954,E2 -503.954} C_VEL
LIN {X 0,Y 608.432,Z 355.325,A -85,B 0,C 180,E1 -506.327,E2 -506.327} C_VEL
LIN {X 0,Y 608.418,Z 355.32,A -85,B 0,C 180,E1 -508.734,E2 -508.734} C_VEL
LIN {X 0,Y 608.391,Z 355.321,A -85,B 0,C 180,E1 -510.976,E2 -510.976} C_VEL
LIN {X 0,Y 608.38,Z 355.321,A -85,B 0,C 180,E1 -513.223,E2 -513.223} C_VEL
LIN {X 0,Y 608.394,Z 355.319,A -85,B 0,C 180,E1 -515.427,E2 -515.427} C_VEL
LIN {X 0,Y 608.437,Z 355.324,A -85,B 0,C 180,E1 -518.307,E2 -518.307} C_VEL
LIN {X 0,Y 608.394,Z 355.319,A -85,B 0,C 180,E1 -521.3,E2 -521.3} C_VEL
LIN {X 0,Y 608.41,Z 355.32,A -85,B 0,C 180,E1 -523.905,E2 -523.905} C_VEL
LIN {X 0,Y 608.427,Z 355.323,A -85,B 0,C 180,E1 -526.643,E2 -526.643} C_VEL
LIN {X 0,Y 608.393,Z 355.319,A -85,B 0,C 180,E1 -529.349,E2 -529.349} C_VEL
LIN {X 0,Y 608.392,Z 355.32,A -85,B 0,C 180,E1 -531.363,E2 -531.363} C_VEL
LIN {X 0,Y 608.417,Z 355.319,A -85,B 0,C 180,E1 -534.033,E2 -534.033} C_VEL
LIN {X 0,Y 608.459,Z 355.319,A -85,B 0,C 180,E1 -536.689,E2 -536.689} C_VEL
LIN {X 0,Y 608.395,Z 355.32,A -85,B 0,C 180,E1 -539.338,E2 -539.338} C_VEL
LIN {X 0,Y 608.407,Z 355.318,A -85,B 0,C 180,E1 -541.324,E2 -541.324} C_VEL
LIN {X 0,Y 608.391,Z 355.32,A -85,B 0,C 180,E1 -543.311,E2 -543.311} C_VEL
LIN {X 0,Y 608.407,Z 355.318,A -85,B 0,C 180,E1 -545.303,E2 -545.303} C_VEL
LIN {X 0,Y 608.401,Z 355.319,A -85,B 0,C 180,E1 -547.3,E2 -547.3} C_VEL
LIN {X 0,Y 608.406,Z 355.318,A -85,B 0,C 180,E1 -549.471,E2 -549.471} C_VEL
LIN {X 0,Y 607.729,Z 355.404,A -85,B 0,C 180,E1 -550.024,E2 -550.024} C_VEL
LIN {X 0,Y 604.877,Z 355.764,A -85,B 0,C 180,E1 -550.921,E2 -550.921} C_VEL
LIN {X 0,Y 602.48,Z 356.06,A -85,B 0,C 180,E1 -551.642,E2 -551.642} C_VEL
LIN {X 0,Y 601.458,Z 356.186,A -85,B 0,C 180,E1 -552.199,E2 -552.199} C_VEL
LIN {X 0,Y 601.379,Z 356.196,A -85,B 0,C 180,E1 -552.388,E2 -552.388} C_VEL
LIN {X 0,Y 601.405,Z 356.197,A -85,B 0,C 180,E1 -554.898,E2 -554.898} C_VEL
LIN {X 0,Y 601.409,Z 356.196,A -85,B 0,C 180,E1 -556.987,E2 -556.987} C_VEL
LIN {X 0,Y 601.365,Z 356.194,A -85,B 0,C 180,E1 -559.811,E2 -559.811} C_VEL
LIN {X 0,Y 601.371,Z 356.194,A -85,B 0,C 180,E1 -561.961,E2 -561.961} C_VEL
LIN {X 0,Y 601.373,Z 356.203,A -85,B 0,C 180,E1 -564.88,E2 -564.88} C_VEL
LIN {X 0,Y 601.373,Z 356.196,A -85,B 0,C 180,E1 -567.358,E2 -567.358} C_VEL
LIN {X 0,Y 601.38,Z 356.195,A -85,B 0,C 180,E1 -569.395,E2 -569.395} C_VEL
LIN {X 0,Y 601.374,Z 356.193,A -85,B 0,C 180,E1 -571.729,E2 -571.729} C_VEL
LIN {X 0,Y 601.4,Z 356.191,A -85,B 0,C 180,E1 -574.12,E2 -574.12} C_VEL
LIN {X 0,Y 601.42,Z 356.191,A -85,B 0,C 180,E1 -577.382,E2 -577.382} C_VEL
LIN {X 0,Y 601.377,Z 356.193,A -85,B 0,C 180,E1 -579.998,E2 -579.998} C_VEL
LIN {X 0,Y 601.397,Z 356.197,A -85,B 0,C 180,E1 -582.672,E2 -582.672} C_VEL
LIN {X 0,Y 601.391,Z 356.195,A -85,B 0,C 180,E1 -585.481,E2 -585.481} C_VEL
LIN {X 0,Y 601.407,Z 356.191,A -85,B 0,C 180,E1 -588.409,E2 -588.409} C_VEL
LIN {X 0,Y 601.394,Z 356.194,A -85,B 0,C 180,E1 -591.534,E2 -591.534} C_VEL
LIN {X 0,Y 601.381,Z 356.194,A -85,B 0,C 180,E1 -593.743,E2 -593.743} C_VEL
LIN {X 0,Y 601.396,Z 356.191,A -85,B 0,C 180,E1 -596.07,E2 -596.07} C_VEL
LIN {X 0,Y 601.411,Z 356.191,A -85,B 0,C 180,E1 -598.547,E2 -598.547} C_VEL
LIN {X 0,Y 601.411,Z 356.197,A -85,B 0,C 180,E1 -601.373,E2 -601.373} C_VEL
LIN {X 0,Y 601.435,Z 356.191,A -85,B 0,C 180,E1 -602.74,E2 -602.74} C_VEL
LIN {X 0,Y 601.991,Z 359.03,A -85,B 0,C 180,E1 -602.802,E2 -602.802} C_VEL
LIN {X 0,Y 601.876,Z 490.637,A -85,B 0,C 180,E1 -604.427,E2 -604.427} C_VEL
LIN {X 0,Y 601.829,Z 506.827,A -85,B 0,C 180,E1 -604.772,E2 -604.772} C_VEL
LIN {X 0,Y 601.773,Z 522.307,A -85,B 0,C 180,E1 -605.256,E2 -605.256} C_VEL
LIN {X 0,Y 601.692,Z 537.115,A -85,B 0,C 180,E1 -605.871,E2 -605.871} C_VEL
LIN {X 0,Y 601.643,Z 551.018,A -85,B 0,C 180,E1 -606.6,E2 -606.6} C_VEL
LIN {X 0,Y 601.587,Z 564.258,A -85,B 0,C 180,E1 -607.451,E2 -607.451} C_VEL
LIN {X 0,Y 601.543,Z 576.573,A -85,B 0,C 180,E1 -608.407,E2 -608.407} C_VEL
LIN {X 0,Y 601.467,Z 588.119,A -85,B 0,C 180,E1 -609.48,E2 -609.48} C_VEL
LIN {X 0,Y 601.442,Z 597.804,A -85,B 0,C 180,E1 -610.548,E2 -610.548} C_VEL
LIN {X 0,Y 601.415,Z 607.201,A -85,B 0,C 180,E1 -611.785,E2 -611.785} C_VEL
LIN {X 0,Y 601.377,Z 614.929,A -85,B 0,C 180,E1 -613.013,E2 -613.013} C_VEL
LIN {X 0,Y 601.339,Z 622.056,A -85,B 0,C 180,E1 -614.407,E2 -614.407} C_VEL
LIN {X 0,Y 601.345,Z 627.578,A -85,B 0,C 180,E1 -615.793,E2 -615.793} C_VEL
LIN {X 0,Y 601.323,Z 631.675,A -85,B 0,C 180,E1 -617.17,E2 -617.17} C_VEL
LIN {X 0,Y 601.319,Z 634.472,A -85,B 0,C 180,E1 -618.54,E2 -618.54} C_VEL
LIN {X 0,Y 601.322,Z 636.05,A -85,B 0,C 180,E1 -619.904,E2 -619.904} C_VEL
LIN {X 0,Y 601.326,Z 636.456,A -85,B 0,C 180,E1 -621.261,E2 -621.261} C_VEL
LIN {X 0,Y 601.32,Z 635.705,A -85,B 0,C 180,E1 -622.614,E2 -622.614} C_VEL
LIN {X 0,Y 601.334,Z 633.792,A -85,B 0,C 180,E1 -623.963,E2 -623.963} C_VEL
LIN {X 0,Y 601.329,Z 630.65,A -85,B 0,C 180,E1 -625.308,E2 -625.308} C_VEL
LIN {X 0,Y 601.343,Z 626.276,A -85,B 0,C 180,E1 -626.65,E2 -626.65} C_VEL
LIN {X 0,Y 601.354,Z 620.579,A -85,B 0,C 180,E1 -627.991,E2 -627.991} C_VEL
LIN {X 0,Y 601.385,Z 613.412,A -85,B 0,C 180,E1 -629.331,E2 -629.331} C_VEL
LIN {X 0,Y 601.412,Z 604.57,A -85,B 0,C 180,E1 -630.67,E2 -630.67} C_VEL
LIN {X 0,Y 601.459,Z 595.203,A -85,B 0,C 180,E1 -631.842,E2 -631.842} C_VEL
LIN {X 0,Y 601.495,Z 583.978,A -85,B 0,C 180,E1 -633.014,E2 -633.014} C_VEL
LIN {X 0,Y 601.557,Z 572.438,A -85,B 0,C 180,E1 -634.02,E2 -634.02} C_VEL
LIN {X 0,Y 601.597,Z 559.775,A -85,B 0,C 180,E1 -634.943,E2 -634.943} C_VEL
LIN {X 0,Y 601.662,Z 547.272,A -85,B 0,C 180,E1 -635.698,E2 -635.698} C_VEL
LIN {X 0,Y 601.729,Z 533.472,A -85,B 0,C 180,E1 -636.382,E2 -636.382} C_VEL
LIN {X 0,Y 601.794,Z 519.163,A -85,B 0,C 180,E1 -636.942,E2 -636.942} C_VEL
LIN {X 0,Y 601.847,Z 504.25,A -85,B 0,C 180,E1 -637.38,E2 -637.38} C_VEL
LIN {X 0,Y 601.862,Z 489.826,A -85,B 0,C 180,E1 -637.675,E2 -637.675} C_VEL
LIN {X 0,Y 601.869,Z 357.931,A -85,B 0,C 180,E1 -639.306,E2 -639.306} C_VEL
LIN {X 0,Y 601.417,Z 356.193,A -85,B 0,C 180,E1 -639.352,E2 -639.352} C_VEL
LIN {X 0,Y 601.37,Z 356.195,A -85,B 0,C 180,E1 -642.143,E2 -642.143} C_VEL
LIN {X 0,Y 601.386,Z 356.202,A -85,B 0,C 180,E1 -644.898,E2 -644.898} C_VEL
LIN {X 0,Y 601.361,Z 356.196,A -85,B 0,C 180,E1 -647.689,E2 -647.689} C_VEL
LIN {X 0,Y 601.367,Z 356.195,A -85,B 0,C 180,E1 -649.81,E2 -649.81} C_VEL
LIN {X 0,Y 601.357,Z 356.196,A -85,B 0,C 180,E1 -651.961,E2 -651.961} C_VEL
LIN {X 0,Y 601.378,Z 356.201,A -85,B 0,C 180,E1 -654.879,E2 -654.879} C_VEL
LIN {X 0,Y 601.395,Z 356.197,A -85,B 0,C 180,E1 -657.358,E2 -657.358} C_VEL
LIN {X 0,Y 601.367,Z 356.194,A -85,B 0,C 180,E1 -660.167,E2 -660.167} C_VEL
LIN {X 0,Y 601.383,Z 356.197,A -85,B 0,C 180,E1 -662.709,E2 -662.709} C_VEL
LIN {X 0,Y 601.366,Z 356.206,A -85,B 0,C 180,E1 -665.107,E2 -665.107} C_VEL
LIN {X 0,Y 601.425,Z 356.193,A -85,B 0,C 180,E1 -667.419,E2 -667.419} C_VEL
LIN {X 0,Y 601.361,Z 356.195,A -85,B 0,C 180,E1 -669.998,E2 -669.998} C_VEL
LIN {X 0,Y 601.355,Z 356.199,A -85,B 0,C 180,E1 -672.674,E2 -672.674} C_VEL
LIN {X 0,Y 601.394,Z 356.197,A -85,B 0,C 180,E1 -675.479,E2 -675.479} C_VEL
LIN {X 0,Y 601.368,Z 356.195,A -85,B 0,C 180,E1 -678.412,E2 -678.412} C_VEL
LIN {X 0,Y 601.375,Z 356.198,A -85,B 0,C 180,E1 -680.87,E2 -680.87} C_VEL
LIN {X 0,Y 601.376,Z 356.197,A -85,B 0,C 180,E1 -683.741,E2 -683.741} C_VEL
LIN {X 0,Y 601.378,Z 356.193,A -85,B 0,C 180,E1 -686.07,E2 -686.07} C_VEL
LIN {X 0,Y 601.373,Z 356.195,A -85,B 0,C 180,E1 -688.551,E2 -688.551} C_VEL
LIN {X 0,Y 601.414,Z 356.199,A -85,B 0,C 180,E1 -691.372,E2 -691.372} C_VEL
LIN {X 0,Y 601.357,Z 356.196,A -85,B 0,C 180,E1 -694.379,E2 -694.379} C_VEL
LIN {X 0,Y 601.35,Z 356.197,A -85,B 0,C 180,E1 -696.587,E2 -696.587} C_VEL
LIN {X 0,Y 601.41,Z 356.198,A -85,B 0,C 180,E1 -699.477,E2 -699.477} C_VEL
LIN {X 0,Y 601.377,Z 356.2,A -85,B 0,C 180,E1 -701.607,E2 -701.607} C_VEL
LIN {X 0,Y 601.406,Z 356.195,A -85,B 0,C 180,E1 -703.712,E2 -703.712} C_VEL
LIN {X 0,Y 601.358,Z 356.195,A -85,B 0,C 180,E1 -706.483,E2 -706.483} C_VEL
LIN {X 0,Y 601.386,Z 356.198,A -85,B 0,C 180,E1 -709.223,E2 -709.223} C_VEL
LIN {X 0,Y 601.375,Z 356.196,A -85,B 0,C 180,E1 -711.938,E2 -711.938} C_VEL
LIN {X 0,Y 601.362,Z 356.198,A -85,B 0,C 180,E1 -713.962,E2 -713.962} C_VEL
LIN {X 0,Y 601.354,Z 356.199,A -85,B 0,C 180,E1 -715.979,E2 -715.979} C_VEL
LIN {X 0,Y 601.378,Z 356.196,A -85,B 0,C 180,E1 -717.991,E2 -717.991} C_VEL
LIN {X 0,Y 601.4,Z 356.194,A -85,B 0,C 180,E1 -720,E2 -720} C_VEL
LIN {X 0,Y 601.381,Z 356.193,A -85,B 0,C 180,E1 -722.679,E2 -722.679} C_VEL
LIN {X 0,Y 601.398,Z 356.198,A -85,B 0,C 180,E1 -725.364,E2 -725.364} C_VEL
LIN {X 0,Y 601.385,Z 356.195,A -85,B 0,C 180,E1 -728.061,E2 -728.061} C_VEL
LIN {X 0,Y 601.38,Z 356.194,A -85,B 0,C 180,E1 -730.996,E2 -730.996} C_VEL
LIN {X 0,Y 601.381,Z 356.202,A -85,B 0,C 180,E1 -733.517,E2 -733.517} C_VEL
LIN {X 0,Y 601.377,Z 356.195,A -85,B 0,C 180,E1 -736.288,E2 -736.288} C_VEL
LIN {X 0,Y 601.388,Z 356.194,A -85,B 0,C 180,E1 -739.1,E2 -739.1} C_VEL
LIN {X 0,Y 601.371,Z 356.2,A -85,B 0,C 180,E1 -741.961,E2 -741.961} C_VEL
LIN {X 0,Y 601.364,Z 356.195,A -85,B 0,C 180,E1 -744.88,E2 -744.88} C_VEL
LIN {X 0,Y 601.381,Z 356.197,A -85,B 0,C 180,E1 -747.358,E2 -747.358} C_VEL
LIN {X 0,Y 601.39,Z 356.196,A -85,B 0,C 180,E1 -750.166,E2 -750.166} C_VEL
LIN {X 0,Y 601.372,Z 356.194,A -85,B 0,C 180,E1 -752.71,E2 -752.71} C_VEL
LIN {X 0,Y 601.356,Z 356.197,A -85,B 0,C 180,E1 -755.108,E2 -755.108} C_VEL
LIN {X 0,Y 601.386,Z 356.197,A -85,B 0,C 180,E1 -757.422,E2 -757.422} C_VEL
LIN {X 0,Y 601.369,Z 356.202,A -85,B 0,C 180,E1 -759.998,E2 -759.998} C_VEL
LIN {X 0,Y 601.346,Z 356.198,A -85,B 0,C 180,E1 -762.585,E2 -762.585} C_VEL
LIN {X 0,Y 601.359,Z 356.197,A -85,B 0,C 180,E1 -764.53,E2 -764.53} C_VEL
LIN {X 0,Y 601.375,Z 356.197,A -85,B 0,C 180,E1 -767.413,E2 -767.413} C_VEL
LIN {X 0,Y 601.387,Z 356.202,A -85,B 0,C 180,E1 -770.004,E2 -770.004} C_VEL
LIN {X 0,Y 601.376,Z 356.195,A -85,B 0,C 180,E1 -772.625,E2 -772.625} C_VEL
LIN {X 0,Y 601.36,Z 356.196,A -85,B 0,C 180,E1 -775.065,E2 -775.065} C_VEL
LIN {X 0,Y 601.406,Z 356.194,A -85,B 0,C 180,E1 -777.483,E2 -777.483} C_VEL
LIN {X 0,Y 601.394,Z 356.328,A -85,B 0,C 180,E1 -780.462,E2 -780.462} C_VEL
LIN {X 0,Y 602.198,Z 360.025,A -85,B 0,C 180,E1 -780.863,E2 -780.863} C_VEL
LIN {X 0,Y 602.132,Z 387.549,A -85,B 0,C 180,E1 -783.484,E2 -783.484} C_VEL
LIN {X 0,Y 601.979,Z 419.266,A -85,B 0,C 180,E1 -786.431,E2 -786.431} C_VEL
LIN {X 0,Y 601.81,Z 452.964,A -85,B 0,C 180,E1 -789.492,E2 -789.492} C_VEL
LIN {X 0,Y 601.732,Z 473.28,A -85,B 0,C 180,E1 -791.308,E2 -791.308} C_VEL
LIN {X 0,Y 602.007,Z 480.142,A -85,B 0,C 180,E1 -791.402,E2 -791.402} C_VEL
LIN {X 0,Y 601.875,Z 641.558,A -85,B 0,C 180,E1 -793.397,E2 -793.397} C_VEL
LIN {X 0,Y 601.813,Z 657.493,A -85,B 0,C 180,E1 -793.745,E2 -793.745} C_VEL
LIN {X 0,Y 601.765,Z 672.052,A -85,B 0,C 180,E1 -794.201,E2 -794.201} C_VEL
LIN {X 0,Y 601.719,Z 685.762,A -85,B 0,C 180,E1 -794.764,E2 -794.764} C_VEL
LIN {X 0,Y 601.657,Z 699.235,A -85,B 0,C 180,E1 -795.455,E2 -795.455} C_VEL
LIN {X 0,Y 601.617,Z 712.45,A -85,B 0,C 180,E1 -796.283,E2 -796.283} C_VEL
LIN {X 0,Y 601.531,Z 724.285,A -85,B 0,C 180,E1 -797.174,E2 -797.174} C_VEL
LIN {X 0,Y 601.488,Z 735.748,A -85,B 0,C 180,E1 -798.201,E2 -798.201} C_VEL
LIN {X 0,Y 601.43,Z 745.389,A -85,B 0,C 180,E1 -799.224,E2 -799.224} C_VEL
LIN {X 0,Y 601.428,Z 754.854,A -85,B 0,C 180,E1 -800.415,E2 -800.415} C_VEL
LIN {X 0,Y 601.368,Z 762.73,A -85,B 0,C 180,E1 -801.6,E2 -801.6} C_VEL
LIN {X 0,Y 601.369,Z 770.087,A -85,B 0,C 180,E1 -802.951,E2 -802.951} C_VEL
LIN {X 0,Y 601.371,Z 775.923,A -85,B 0,C 180,E1 -804.299,E2 -804.299} C_VEL
LIN {X 0,Y 601.33,Z 779.383,A -85,B 0,C 180,E1 -805.307,E2 -805.307} C_VEL
LIN {X 0,Y 601.337,Z 782.886,A -85,B 0,C 180,E1 -806.65,E2 -806.65} C_VEL
LIN {X 0,Y 601.339,Z 785.192,A -85,B 0,C 180,E1 -807.99,E2 -807.99} C_VEL
LIN {X 0,Y 601.337,Z 786.35,A -85,B 0,C 180,E1 -809.33,E2 -809.33} C_VEL
LIN {X 0,Y 601.337,Z 786.35,A -85,B 0,C 180,E1 -810.669,E2 -810.669} C_VEL
LIN {X 0,Y 601.339,Z 785.192,A -85,B 0,C 180,E1 -812.009,E2 -812.009} C_VEL
LIN {X 0,Y 601.337,Z 782.886,A -85,B 0,C 180,E1 -813.35,E2 -813.35} C_VEL
LIN {X 0,Y 601.33,Z 779.384,A -85,B 0,C 180,E1 -814.692,E2 -814.692} C_VEL
LIN {X 0,Y 601.352,Z 774.609,A -85,B 0,C 180,E1 -816.037,E2 -816.037} C_VEL
LIN {X 0,Y 601.382,Z 768.428,A -85,B 0,C 180,E1 -817.385,E2 -817.385} C_VEL
LIN {X 0,Y 601.387,Z 760.656,A -85,B 0,C 180,E1 -818.738,E2 -818.738} C_VEL
LIN {X 0,Y 601.427,Z 752.374,A -85,B 0,C 180,E1 -819.925,E2 -819.925} C_VEL
LIN {X 0,Y 601.46,Z 741.935,A -85,B 0,C 180,E1 -821.164,E2 -821.164} C_VEL
LIN {X 0,Y 601.513,Z 732.198,A -85,B 0,C 180,E1 -822.14,E2 -822.14} C_VEL
LIN {X 0,Y 601.57,Z 720.023,A -85,B 0,C 180,E1 -823.168,E2 -823.168} C_VEL
LIN {X 0,Y 601.605,Z 708.087,A -85,B 0,C 180,E1 -824.011,E2 -824.011} C_VEL
LIN {X 0,Y 601.649,Z 694.539,A -85,B 0,C 180,E1 -824.804,E2 -824.804} C_VEL
LIN {X 0,Y 601.761,Z 679.858,A -85,B 0,C 180,E1 -825.495,E2 -825.495} C_VEL
LIN {X 0,Y 601.782,Z 665.638,A -85,B 0,C 180,E1 -826.015,E2 -826.015} C_VEL
LIN {X 0,Y 601.856,Z 650.708,A -85,B 0,C 180,E1 -826.42,E2 -826.42} C_VEL
LIN {X 0,Y 601.866,Z 635.744,A -85,B 0,C 180,E1 -826.689,E2 -826.689} C_VEL
LIN {X 0,Y 601.929,Z 474.583,A -85,B 0,C 180,E1 -828.67,E2 -828.67} C_VEL
LIN {X 0,Y 601.721,Z 472.951,A -85,B 0,C 180,E1 -828.72,E2 -828.72} C_VEL
LIN {X 0,Y 601.836,Z 443.059,A -85,B 0,C 180,E1 -831.402,E2 -831.402} C_VEL
LIN {X 0,Y 601.998,Z 411.727,A -85,B 0,C 180,E1 -834.264,E2 -834.264} C_VEL
LIN {X 0,Y 602.142,Z 381.608,A -85,B 0,C 180,E1 -837.076,E2 -837.076} C_VEL
LIN {X 0,Y 602.215,Z 360.872,A -85,B 0,C 180,E1 -839.055,E2 -839.055} C_VEL
LIN {X 0,Y 601.39,Z 356.2,A -85,B 0,C 180,E1 -839.562,E2 -839.562} C_VEL
LIN {X 0,Y 601.406,Z 356.194,A -85,B 0,C 180,E1 -842.516,E2 -842.516} C_VEL
LIN {X 0,Y 601.349,Z 356.197,A -85,B 0,C 180,E1 -845.106,E2 -845.106} C_VEL
LIN {X 0,Y 601.375,Z 356.195,A -85,B 0,C 180,E1 -847.422,E2 -847.422} C_VEL
LIN {X 0,Y 601.384,Z 356.202,A -85,B 0,C 180,E1 -849.996,E2 -849.996} C_VEL
LIN {X 0,Y 601.365,Z 356.197,A -85,B 0,C 180,E1 -852.673,E2 -852.673} C_VEL
LIN {X 0,Y 601.356,Z 356.196,A -85,B 0,C 180,E1 -855.476,E2 -855.476} C_VEL
LIN {X 0,Y 601.395,Z 356.198,A -85,B 0,C 180,E1 -858.408,E2 -858.408} C_VEL
LIN {X 0,Y 601.369,Z 356.195,A -85,B 0,C 180,E1 -860.87,E2 -860.87} C_VEL
LIN {X 0,Y 601.371,Z 356.197,A -85,B 0,C 180,E1 -863.741,E2 -863.741} C_VEL
LIN {X 0,Y 601.368,Z 356.198,A -85,B 0,C 180,E1 -866.683,E2 -866.683} C_VEL
LIN {X 0,Y 601.369,Z 356.195,A -85,B 0,C 180,E1 -869.055,E2 -869.055} C_VEL
LIN {X 0,Y 601.344,Z 356.198,A -85,B 0,C 180,E1 -871.369,E2 -871.369} C_VEL
LIN {X 0,Y 601.396,Z 356.198,A -85,B 0,C 180,E1 -874.132,E2 -874.132} C_VEL
LIN {X 0,Y 601.36,Z 356.202,A -85,B 0,C 180,E1 -876.587,E2 -876.587} C_VEL
LIN {X 0,Y 601.37,Z 356.194,A -85,B 0,C 180,E1 -879.476,E2 -879.476} C_VEL
LIN {X 0,Y 601.344,Z 356.198,A -85,B 0,C 180,E1 -881.606,E2 -881.606} C_VEL
LIN {X 0,Y 601.376,Z 356.204,A -85,B 0,C 180,E1 -884.408,E2 -884.408} C_VEL
LIN {X 0,Y 601.343,Z 356.199,A -85,B 0,C 180,E1 -887.17,E2 -887.17} C_VEL
LIN {X 0,Y 601.356,Z 356.197,A -85,B 0,C 180,E1 -889.223,E2 -889.223} C_VEL
LIN {X 0,Y 601.381,Z 356.195,A -85,B 0,C 180,E1 -891.939,E2 -891.939} C_VEL
LIN {X 0,Y 601.403,Z 356.199,A -85,B 0,C 180,E1 -894.636,E2 -894.636} C_VEL
LIN {X 0,Y 601.382,Z 356.193,A -85,B 0,C 180,E1 -897.321,E2 -897.321} C_VEL
LIN {X 0,Y 601.398,Z 356.193,A -85,B 0,C 180,E1 -900,E2 -900} C_VEL
LIN {X 0,Y 601.436,Z 356.196,A -85,B 0,C 180,E1 -902.679,E2 -902.679} C_VEL
LIN {X 0,Y 601.373,Z 356.194,A -85,B 0,C 180,E1 -905.365,E2 -905.365} C_VEL
LIN {X 0,Y 601.353,Z 356.196,A -85,B 0,C 180,E1 -907.386,E2 -907.386} C_VEL
LIN {X 0,Y 601.362,Z 356.195,A -85,B 0,C 180,E1 -909.468,E2 -909.468} C_VEL
LIN {X 0,Y 601.383,Z 356.195,A -85,B 0,C 180,E1 -912.143,E2 -912.143} C_VEL
LIN {X 0,Y 601.379,Z 356.196,A -85,B 0,C 180,E1 -912.388,E2 -912.388} C_VEL
LIN {X 0,Y 600.723,Z 356.283,A -85,B 0,C 180,E1 -912.947,E2 -912.947} C_VEL
LIN {X 0,Y 597.877,Z 356.637,A -85,B 0,C 180,E1 -913.855,E2 -913.855} C_VEL
LIN {X 0,Y 595.461,Z 356.938,A -85,B 0,C 180,E1 -914.585,E2 -914.585} C_VEL
LIN {X 0,Y 594.415,Z 357.064,A -85,B 0,C 180,E1 -915.149,E2 -915.149} C_VEL
LIN {X 0,Y 594.326,Z 357.073,A -85,B 0,C 180,E1 -915.34,E2 -915.34} C_VEL
LIN {X 0,Y 594.362,Z 357.07,A -85,B 0,C 180,E1 -917.194,E2 -917.194} C_VEL
LIN {X 0,Y 594.345,Z 357.07,A -85,B 0,C 180,E1 -920.055,E2 -920.055} C_VEL
LIN {X 0,Y 594.337,Z 357.078,A -85,B 0,C 180,E1 -922.969,E2 -922.969} C_VEL
LIN {X 0,Y 594.333,Z 357.074,A -85,B 0,C 180,E1 -925.195,E2 -925.195} C_VEL
LIN {X 0,Y 594.328,Z 357.072,A -85,B 0,C 180,E1 -927.519,E2 -927.519} C_VEL
LIN {X 0,Y 594.34,Z 357.07,A -85,B 0,C 180,E1 -929.779,E2 -929.779} C_VEL
LIN {X 0,Y 594.345,Z 357.069,A -85,B 0,C 180,E1 -932.149,E2 -932.149} C_VEL
LIN {X 0,Y 594.37,Z 357.072,A -85,B 0,C 180,E1 -934.581,E2 -934.581} C_VEL
LIN {X 0,Y 594.37,Z 357.067,A -85,B 0,C 180,E1 -937.608,E2 -937.608} C_VEL
LIN {X 0,Y 594.348,Z 357.073,A -85,B 0,C 180,E1 -940.569,E2 -940.569} C_VEL
LIN {X 0,Y 594.341,Z 357.074,A -85,B 0,C 180,E1 -943.302,E2 -943.302} C_VEL
LIN {X 0,Y 594.351,Z 357.069,A -85,B 0,C 180,E1 -946.163,E2 -946.163} C_VEL
LIN {X 0,Y 594.369,Z 357.074,A -85,B 0,C 180,E1 -949.179,E2 -949.179} C_VEL
LIN {X 0,Y 594.361,Z 357.067,A -85,B 0,C 180,E1 -952.059,E2 -952.059} C_VEL
LIN {X 0,Y 594.325,Z 357.076,A -85,B 0,C 180,E1 -954.681,E2 -954.681} C_VEL
LIN {X 0,Y 594.369,Z 357.077,A -85,B 0,C 180,E1 -957.091,E2 -957.091} C_VEL
LIN {X 0,Y 594.345,Z 357.072,A -85,B 0,C 180,E1 -959.679,E2 -959.679} C_VEL
LIN {X 0,Y 594.327,Z 357.075,A -85,B 0,C 180,E1 -961.772,E2 -961.772} C_VEL
LIN {X 0,Y 594.355,Z 357.071,A -85,B 0,C 180,E1 -962.525,E2 -962.525} C_VEL
LIN {X 0,Y 595.25,Z 360.624,A -85,B 0,C 180,E1 -962.608,E2 -962.608} C_VEL
LIN {X 0,Y 595.088,Z 490.6,A -85,B 0,C 180,E1 -964.231,E2 -964.231} C_VEL
LIN {X 0,Y 595.032,Z 505.894,A -85,B 0,C 180,E1 -964.557,E2 -964.557} C_VEL
LIN {X 0,Y 594.93,Z 520.93,A -85,B 0,C 180,E1 -965.02,E2 -965.02} C_VEL
LIN {X 0,Y 594.845,Z 535.599,A -85,B 0,C 180,E1 -965.621,E2 -965.621} C_VEL
LIN {X 0,Y 594.725,Z 548.96,A -85,B 0,C 180,E1 -966.311,E2 -966.311} C_VEL
LIN {X 0,Y 594.659,Z 561.805,A -85,B 0,C 180,E1 -967.12,E2 -967.12} C_VEL
LIN {X 0,Y 594.563,Z 574.081,A -85,B 0,C 180,E1 -968.049,E2 -968.049} C_VEL
LIN {X 0,Y 594.456,Z 585.344,A -85,B 0,C 180,E1 -969.065,E2 -969.065} C_VEL
LIN {X 0,Y 594.402,Z 595.286,A -85,B 0,C 180,E1 -970.128,E2 -970.128} C_VEL
LIN {X 0,Y 594.338,Z 605.127,A -85,B 0,C 180,E1 -971.382,E2 -971.382} C_VEL
LIN {X 0,Y 594.316,Z 613.221,A -85,B 0,C 180,E1 -972.628,E2 -972.628} C_VEL
LIN {X 0,Y 594.298,Z 619.867,A -85,B 0,C 180,E1 -973.866,E2 -973.866} C_VEL
LIN {X 0,Y 594.262,Z 625.906,A -85,B 0,C 180,E1 -975.27,E2 -975.27} C_VEL
LIN {X 0,Y 594.255,Z 629.454,A -85,B 0,C 180,E1 -976.319,E2 -976.319} C_VEL
LIN {X 0,Y 594.236,Z 633.001,A -85,B 0,C 180,E1 -977.709,E2 -977.709} C_VEL
LIN {X 0,Y 594.239,Z 635.286,A -85,B 0,C 180,E1 -979.093,E2 -979.093} C_VEL
LIN {X 0,Y 594.248,Z 636.374,A -85,B 0,C 180,E1 -980.47,E2 -980.47} C_VEL
LIN {X 0,Y 594.226,Z 636.298,A -85,B 0,C 180,E1 -981.841,E2 -981.841} C_VEL
LIN {X 0,Y 594.272,Z 635.04,A -85,B 0,C 180,E1 -983.209,E2 -983.209} C_VEL
LIN {X 0,Y 594.262,Z 632.599,A -85,B 0,C 180,E1 -984.571,E2 -984.571} C_VEL
LIN {X 0,Y 594.259,Z 628.955,A -85,B 0,C 180,E1 -985.931,E2 -985.931} C_VEL
LIN {X 0,Y 594.243,Z 624.049,A -85,B 0,C 180,E1 -987.289,E2 -987.289} C_VEL
LIN {X 0,Y 594.288,Z 617.761,A -85,B 0,C 180,E1 -988.645,E2 -988.645} C_VEL
LIN {X 0,Y 594.348,Z 609.919,A -85,B 0,C 180,E1 -990,E2 -990} C_VEL
LIN {X 0,Y 594.387,Z 601.612,A -85,B 0,C 180,E1 -991.186,E2 -991.186} C_VEL
LIN {X 0,Y 594.432,Z 591.664,A -85,B 0,C 180,E1 -992.372,E2 -992.372} C_VEL
LIN {X 0,Y 594.545,Z 581.56,A -85,B 0,C 180,E1 -993.389,E2 -993.389} C_VEL
LIN {X 0,Y 594.591,Z 569.541,A -85,B 0,C 180,E1 -994.406,E2 -994.406} C_VEL
LIN {X 0,Y 594.678,Z 557.595,A -85,B 0,C 180,E1 -995.255,E2 -995.255} C_VEL
LIN {X 0,Y 594.784,Z 544.616,A -85,B 0,C 180,E1 -996.02,E2 -996.02} C_VEL
LIN {X 0,Y 594.868,Z 530.152,A -85,B 0,C 180,E1 -996.711,E2 -996.711} C_VEL
LIN {X 0,Y 594.973,Z 515.523,A -85,B 0,C 180,E1 -997.252,E2 -997.252} C_VEL
LIN {X 0,Y 595.047,Z 500.737,A -85,B 0,C 180,E1 -997.657,E2 -997.657} C_VEL
LIN {X 0,Y 595.032,Z 485.54,A -85,B 0,C 180,E1 -997.935,E2 -997.935} C_VEL
LIN {X 0,Y 595.135,Z 359.535,A -85,B 0,C 180,E1 -999.5,E2 -999.5} C_VEL
LIN {X 0,Y 594.332,Z 357.074,A -85,B 0,C 180,E1 -999.572,E2 -999.572} C_VEL
LIN {X 0,Y 594.367,Z 357.069,A -85,B 0,C 180,E1 -1001.596,E2 -1001.596} C_VEL
LIN {X 0,Y 594.325,Z 357.074,A -85,B 0,C 180,E1 -1004.379,E2 -1004.379} C_VEL
LIN {X 0,Y 594.323,Z 357.08,A -85,B 0,C 180,E1 -1007.195,E2 -1007.195} C_VEL
LIN {X 0,Y 594.349,Z 357.074,A -85,B 0,C 180,E1 -1009.335,E2 -1009.335} C_VEL
LIN {X 0,Y 594.334,Z 357.074,A -85,B 0,C 180,E1 -1011.504,E2 -1011.504} C_VEL
LIN {X 0,Y 594.339,Z 357.072,A -85,B 0,C 180,E1 -1014.448,E2 -1014.448} C_VEL
LIN {X 0,Y 594.336,Z 357.075,A -85,B 0,C 180,E1 -1017.462,E2 -1017.462} C_VEL
LIN {X 0,Y 594.343,Z 357.069,A -85,B 0,C 180,E1 -1020.32,E2 -1020.32} C_VEL
LIN {X 0,Y 594.335,Z 357.079,A -85,B 0,C 180,E1 -1022.952,E2 -1022.952} C_VEL
LIN {X 0,Y 594.3,Z 357.081,A -85,B 0,C 180,E1 -1025.412,E2 -1025.412} C_VEL
LIN {X 0,Y 594.339,Z 357.071,A -85,B 0,C 180,E1 -1027.943,E2 -1027.943} C_VEL
LIN {X 0,Y 594.353,Z 357.073,A -85,B 0,C 180,E1 -1030.819,E2 -1030.819} C_VEL
LIN {X 0,Y 594.329,Z 357.073,A -85,B 0,C 180,E1 -1033.835,E2 -1033.835} C_VEL
LIN {X 0,Y 594.332,Z 357.074,A -85,B 0,C 180,E1 -1036.697,E2 -1036.697} C_VEL
LIN {X 0,Y 594.346,Z 357.077,A -85,B 0,C 180,E1 -1039.431,E2 -1039.431} C_VEL
LIN {X 0,Y 594.336,Z 357.07,A -85,B 0,C 180,E1 -1042.397,E2 -1042.397} C_VEL
LIN {X 0,Y 594.36,Z 357.075,A -85,B 0,C 180,E1 -1045.418,E2 -1045.418} C_VEL
LIN {X 0,Y 594.342,Z 357.07,A -85,B 0,C 180,E1 -1048.361,E2 -1048.361} C_VEL
LIN {X 0,Y 594.366,Z 357.073,A -85,B 0,C 180,E1 -1051.043,E2 -1051.043} C_VEL
LIN {X 0,Y 594.329,Z 357.072,A -85,B 0,C 180,E1 -1054.053,E2 -1054.053} C_VEL
LIN {X 0,Y 594.333,Z 357.07,A -85,B 0,C 180,E1 -1056.293,E2 -1056.293} C_VEL
LIN {X 0,Y 594.39,Z 357.072,A -85,B 0,C 180,E1 -1059.224,E2 -1059.224} C_VEL
LIN {X 0,Y 594.307,Z 357.075,A -85,B 0,C 180,E1 -1062.093,E2 -1062.093} C_VEL
LIN {X 0,Y 594.315,Z 357.073,A -85,B 0,C 180,E1 -1064.217,E2 -1064.217} C_VEL
LIN {X 0,Y 594.332,Z 357.074,A -85,B 0,C 180,E1 -1067.016,E2 -1067.016} C_VEL
LIN {X 0,Y 594.321,Z 357.076,A -85,B 0,C 180,E1 -1069.783,E2 -1069.783} C_VEL
LIN {X 0,Y 594.332,Z 357.075,A -85,B 0,C 180,E1 -1071.842,E2 -1071.842} C_VEL
LIN {X 0,Y 594.321,Z 357.076,A -85,B 0,C 180,E1 -1073.89,E2 -1073.89} C_VEL
LIN {X 0,Y 594.311,Z 357.077,A -85,B 0,C 180,E1 -1075.931,E2 -1075.931} C_VEL
LIN {X 0,Y 594.352,Z 357.071,A -85,B 0,C 180,E1 -1077.967,E2 -1077.967} C_VEL
LIN {X 0,Y 594.372,Z 357.069,A -85,B 0,C 180,E1 -1080,E2 -1080} C_VEL
LIN {X 0,Y 594.352,Z 357.068,A -85,B 0,C 180,E1 -1082.711,E2 -1082.711} C_VEL
LIN {X 0,Y 594.362,Z 357.075,A -85,B 0,C 180,E1 -1085.428,E2 -1085.428} C_VEL
LIN {X 0,Y 594.335,Z 357.072,A -85,B 0,C 180,E1 -1088.158,E2 -1088.158} C_VEL
LIN {X 0,Y 594.352,Z 357.071,A -85,B 0,C 180,E1 -1091.061,E2 -1091.061} C_VEL
LIN {X 0,Y 594.341,Z 357.072,A -85,B 0,C 180,E1 -1094.16,E2 -1094.16} C_VEL
LIN {X 0,Y 594.307,Z 357.074,A -85,B 0,C 180,E1 -1096.695,E2 -1096.695} C_VEL
LIN {X 0,Y 594.341,Z 357.074,A -85,B 0,C 180,E1 -1099.335,E2 -1099.335} C_VEL
LIN {X 0,Y 594.334,Z 357.078,A -85,B 0,C 180,E1 -1101.504,E2 -1101.504} C_VEL
LIN {X 0,Y 594.331,Z 357.072,A -85,B 0,C 180,E1 -1104.448,E2 -1104.448} C_VEL
LIN {X 0,Y 594.339,Z 357.07,A -85,B 0,C 180,E1 -1106.702,E2 -1106.702} C_VEL
LIN {X 0,Y 594.346,Z 357.08,A -85,B 0,C 180,E1 -1109.778,E2 -1109.778} C_VEL
LIN {X 0,Y 594.329,Z 357.075,A -85,B 0,C 180,E1 -1112.149,E2 -1112.149} C_VEL
LIN {X 0,Y 594.34,Z 357.07,A -85,B 0,C 180,E1 -1114.583,E2 -1114.583} C_VEL
LIN {X 0,Y 594.346,Z 357.077,A -85,B 0,C 180,E1 -1117.604,E2 -1117.604} C_VEL
LIN {X 0,Y 594.342,Z 357.071,A -85,B 0,C 180,E1 -1120.569,E2 -1120.569} C_VEL
LIN {X 0,Y 594.328,Z 357.074,A -85,B 0,C 180,E1 -1123.303,E2 -1123.303} C_VEL
LIN {X 0,Y 594.335,Z 357.077,A -85,B 0,C 180,E1 -1126.164,E2 -1126.164} C_VEL
LIN {X 0,Y 594.348,Z 357.069,A -85,B 0,C 180,E1 -1128.534,E2 -1128.534} C_VEL
LIN {X 0,Y 594.355,Z 357.07,A -85,B 0,C 180,E1 -1131.299,E2 -1131.299} C_VEL
LIN {X 0,Y 594.336,Z 357.079,A -85,B 0,C 180,E1 -1133.755,E2 -1133.755} C_VEL
LIN {X 0,Y 594.348,Z 357.076,A -85,B 0,C 180,E1 -1136.238,E2 -1136.238} C_VEL
LIN {X 0,Y 594.32,Z 357.076,A -85,B 0,C 180,E1 -1138.647,E2 -1138.647} C_VEL
LIN {X 0,Y 594.4,Z 357.151,A -85,B 0,C 180,E1 -1140.16,E2 -1140.16} C_VEL
LIN {X 0,Y 595.56,Z 361.772,A -85,B 0,C 180,E1 -1140.677,E2 -1140.677} C_VEL
LIN {X 0,Y 595.469,Z 385.567,A -85,B 0,C 180,E1 -1142.974,E2 -1142.974} C_VEL
LIN {X 0,Y 595.24,Z 415.301,A -85,B 0,C 180,E1 -1145.777,E2 -1145.777} C_VEL
LIN {X 0,Y 595.015,Z 445.035,A -85,B 0,C 180,E1 -1148.522,E2 -1148.522} C_VEL
LIN {X 0,Y 594.836,Z 473.226,A -85,B 0,C 180,E1 -1151.08,E2 -1151.08} C_VEL
LIN {X 0,Y 595.305,Z 477.314,A -85,B 0,C 180,E1 -1151.149,E2 -1151.149} C_VEL
LIN {X 0,Y 595.082,Z 641.36,A -85,B 0,C 180,E1 -1153.199,E2 -1153.199} C_VEL
LIN {X 0,Y 595.017,Z 656.716,A -85,B 0,C 180,E1 -1153.533,E2 -1153.533} C_VEL
LIN {X 0,Y 594.931,Z 672.051,A -85,B 0,C 180,E1 -1154.015,E2 -1154.015} C_VEL
LIN {X 0,Y 594.856,Z 685.765,A -85,B 0,C 180,E1 -1154.584,E2 -1154.584} C_VEL
LIN {X 0,Y 594.731,Z 699.237,A -85,B 0,C 180,E1 -1155.282,E2 -1155.282} C_VEL
LIN {X 0,Y 594.68,Z 711.793,A -85,B 0,C 180,E1 -1156.075,E2 -1156.075} C_VEL
LIN {X 0,Y 594.559,Z 724.286,A -85,B 0,C 180,E1 -1157.021,E2 -1157.021} C_VEL
LIN {X 0,Y 594.465,Z 735.749,A -85,B 0,C 180,E1 -1158.06,E2 -1158.06} C_VEL
LIN {X 0,Y 594.388,Z 745.389,A -85,B 0,C 180,E1 -1159.095,E2 -1159.095} C_VEL
LIN {X 0,Y 594.366,Z 754.855,A -85,B 0,C 180,E1 -1160.3,E2 -1160.3} C_VEL
LIN {X 0,Y 594.311,Z 762.73,A -85,B 0,C 180,E1 -1161.499,E2 -1161.499} C_VEL
LIN {X 0,Y 594.292,Z 770.088,A -85,B 0,C 180,E1 -1162.867,E2 -1162.867} C_VEL
LIN {X 0,Y 594.296,Z 775.924,A -85,B 0,C 180,E1 -1164.231,E2 -1164.231} C_VEL
LIN {X 0,Y 594.232,Z 779.383,A -85,B 0,C 180,E1 -1165.251,E2 -1165.251} C_VEL
LIN {X 0,Y 594.257,Z 782.886,A -85,B 0,C 180,E1 -1166.61,E2 -1166.61} C_VEL
LIN {X 0,Y 594.238,Z 785.192,A -85,B 0,C 180,E1 -1167.966,E2 -1167.966} C_VEL
LIN {X 0,Y 594.237,Z 786.35,A -85,B 0,C 180,E1 -1169.322,E2 -1169.322} C_VEL
LIN {X 0,Y 594.237,Z 786.35,A -85,B 0,C 180,E1 -1170.677,E2 -1170.677} C_VEL
LIN {X 0,Y 594.238,Z 785.192,A -85,B 0,C 180,E1 -1172.033,E2 -1172.033} C_VEL
LIN {X 0,Y 594.257,Z 782.887,A -85,B 0,C 180,E1 -1173.39,E2 -1173.39} C_VEL
LIN {X 0,Y 594.232,Z 779.385,A -85,B 0,C 180,E1 -1174.749,E2 -1174.749} C_VEL
LIN {X 0,Y 594.275,Z 774.61,A -85,B 0,C 180,E1 -1176.109,E2 -1176.109} C_VEL
LIN {X 0,Y 594.296,Z 768.427,A -85,B 0,C 180,E1 -1177.474,E2 -1177.474} C_VEL
LIN {X 0,Y 594.331,Z 760.655,A -85,B 0,C 180,E1 -1178.842,E2 -1178.842} C_VEL
LIN {X 0,Y 594.387,Z 752.374,A -85,B 0,C 180,E1 -1180.043,E2 -1180.043} C_VEL
LIN {X 0,Y 594.433,Z 742.561,A -85,B 0,C 180,E1 -1181.231,E2 -1181.231} C_VEL
LIN {X 0,Y 594.53,Z 732.198,A -85,B 0,C 180,E1 -1182.285,E2 -1182.285} C_VEL
LIN {X 0,Y 594.581,Z 720.024,A -85,B 0,C 180,E1 -1183.325,E2 -1183.325} C_VEL
LIN {X 0,Y 594.693,Z 708.084,A -85,B 0,C 180,E1 -1184.177,E2 -1184.177} C_VEL
LIN {X 0,Y 594.75,Z 694.536,A -85,B 0,C 180,E1 -1184.98,E2 -1184.98} C_VEL
LIN {X 0,Y 594.902,Z 679.856,A -85,B 0,C 180,E1 -1185.678,E2 -1185.678} C_VEL
LIN {X 0,Y 594.961,Z 665.638,A -85,B 0,C 180,E1 -1186.204,E2 -1186.204} C_VEL
LIN {X 0,Y 595.048,Z 651.142,A -85,B 0,C 180,E1 -1186.602,E2 -1186.602} C_VEL
LIN {X 0,Y 595.067,Z 635.744,A -85,B 0,C 180,E1 -1186.886,E2 -1186.886} C_VEL
LIN {X 0,Y 595.286,Z 476.046,A -85,B 0,C 180,E1 -1188.867,E2 -1188.867} C_VEL
LIN {X 0,Y 594.865,Z 473.209,A -85,B 0,C 180,E1 -1188.921,E2 -1188.921} C_VEL
LIN {X 0,Y 595.035,Z 443.059,A -85,B 0,C 180,E1 -1191.659,E2 -1191.659} C_VEL
LIN {X 0,Y 595.265,Z 412.632,A -85,B 0,C 180,E1 -1194.472,E2 -1194.472} C_VEL
LIN {X 0,Y 595.48,Z 381.608,A -85,B 0,C 180,E1 -1197.405,E2 -1197.405} C_VEL
LIN {X 0,Y 595.605,Z 363.315,A -85,B 0,C 180,E1 -1199.17,E2 -1199.17} C_VEL
LIN {X 0,Y 595.033,Z 359.616,A -85,B 0,C 180,E1 -1199.563,E2 -1199.563} C_VEL
LIN {X 0,Y 594.386,Z 357.073,A -85,B 0,C 180,E1 -1199.862,E2 -1199.862} C_VEL
LIN {X 0,Y 594.364,Z 357.068,A -85,B 0,C 180,E1 -1202.95,E2 -1202.95} C_VEL
LIN {X 0,Y 594.302,Z 357.076,A -85,B 0,C 180,E1 -1205.411,E2 -1205.411} C_VEL
LIN {X 0,Y 594.359,Z 357.076,A -85,B 0,C 180,E1 -1207.941,E2 -1207.941} C_VEL
LIN {X 0,Y 594.342,Z 357.071,A -85,B 0,C 180,E1 -1210.818,E2 -1210.818} C_VEL
LIN {X 0,Y 594.33,Z 357.072,A -85,B 0,C 180,E1 -1213.301,E2 -1213.301} C_VEL
LIN {X 0,Y 594.324,Z 357.081,A -85,B 0,C 180,E1 -1216.163,E2 -1216.163} C_VEL
LIN {X 0,Y 594.352,Z 357.073,A -85,B 0,C 180,E1 -1218.534,E2 -1218.534} C_VEL
LIN {X 0,Y 594.34,Z 357.07,A -85,B 0,C 180,E1 -1221.299,E2 -1221.299} C_VEL
LIN {X 0,Y 594.326,Z 357.075,A -85,B 0,C 180,E1 -1223.754,E2 -1223.754} C_VEL
LIN {X 0,Y 594.337,Z 357.081,A -85,B 0,C 180,E1 -1226.236,E2 -1226.236} C_VEL
LIN {X 0,Y 594.342,Z 357.074,A -85,B 0,C 180,E1 -1228.648,E2 -1228.648} C_VEL
LIN {X 0,Y 594.318,Z 357.074,A -85,B 0,C 180,E1 -1231.05,E2 -1231.05} C_VEL
LIN {X 0,Y 594.352,Z 357.074,A -85,B 0,C 180,E1 -1234.055,E2 -1234.055} C_VEL
LIN {X 0,Y 594.308,Z 357.076,A -85,B 0,C 180,E1 -1237.031,E2 -1237.031} C_VEL
LIN {X 0,Y 594.352,Z 357.069,A -85,B 0,C 180,E1 -1239.223,E2 -1239.223} C_VEL
LIN {X 0,Y 594.305,Z 357.08,A -85,B 0,C 180,E1 -1242.094,E2 -1242.094} C_VEL
LIN {X 0,Y 594.318,Z 357.076,A -85,B 0,C 180,E1 -1244.921,E2 -1244.921} C_VEL
LIN {X 0,Y 594.324,Z 357.073,A -85,B 0,C 180,E1 -1247.711,E2 -1247.711} C_VEL
LIN {X 0,Y 594.33,Z 357.082,A -85,B 0,C 180,E1 -1250.471,E2 -1250.471} C_VEL
LIN {X 0,Y 594.317,Z 357.073,A -85,B 0,C 180,E1 -1253.362,E2 -1253.362} C_VEL
LIN {X 0,Y 594.311,Z 357.075,A -85,B 0,C 180,E1 -1255.931,E2 -1255.931} C_VEL
LIN {X 0,Y 594.367,Z 357.076,A -85,B 0,C 180,E1 -1258.645,E2 -1258.645} C_VEL
LIN {X 0,Y 594.408,Z 357.07,A -85,B 0,C 180,E1 -1260.678,E2 -1260.678} C_VEL
LIN {X 0,Y 594.298,Z 357.076,A -85,B 0,C 180,E1 -1263.39,E2 -1263.39} C_VEL
LIN {X 0,Y 594.339,Z 357.069,A -85,B 0,C 180,E1 -1265.428,E2 -1265.428} C_VEL
LIN {X 0,Y 594.325,Z 357.07,A -85,B 0,C 180,E1 -1267.474,E2 -1267.474} C_VEL
LIN {X 0,Y 594.315,Z 357.073,A -85,B 0,C 180,E1 -1269.53,E2 -1269.53} C_VEL
LIN {X 0,Y 594.351,Z 357.069,A -85,B 0,C 180,E1 -1271.597,E2 -1271.597} C_VEL
LIN {X 0,Y 594.365,Z 357.071,A -85,B 0,C 180,E1 -1274.378,E2 -1274.378} C_VEL
LIN {X 0,Y 594.326,Z 357.073,A -85,B 0,C 180,E1 -1275.34,E2 -1275.34} C_VEL
LIN {X 0,Y 593.644,Z 357.158,A -85,B 0,C 180,E1 -1275.905,E2 -1275.905} C_VEL
LIN {X 0,Y 590.771,Z 357.524,A -85,B 0,C 180,E1 -1276.823,E2 -1276.823} C_VEL
LIN {X 0,Y 588.365,Z 357.819,A -85,B 0,C 180,E1 -1277.562,E2 -1277.562} C_VEL
LIN {X 0,Y 587.352,Z 357.942,A -85,B 0,C 180,E1 -1278.132,E2 -1278.132} C_VEL
LIN {X 0,Y 587.281,Z 357.952,A -85,B 0,C 180,E1 -1278.325,E2 -1278.325} C_VEL
LIN {X 0,Y 587.317,Z 357.95,A -85,B 0,C 180,E1 -1281.038,E2 -1281.038} C_VEL
LIN {X 0,Y 587.285,Z 357.949,A -85,B 0,C 180,E1 -1284.009,E2 -1284.009} C_VEL
LIN {X 0,Y 587.276,Z 357.952,A -85,B 0,C 180,E1 -1286.282,E2 -1286.282} C_VEL
LIN {X 0,Y 587.333,Z 357.949,A -85,B 0,C 180,E1 -1289.134,E2 -1289.134} C_VEL
LIN {X 0,Y 587.327,Z 357.942,A -85,B 0,C 180,E1 -1291.836,E2 -1291.836} C_VEL
LIN {X 0,Y 587.328,Z 357.946,A -85,B 0,C 180,E1 -1294.347,E2 -1294.347} C_VEL
LIN {X 0,Y 587.337,Z 357.95,A -85,B 0,C 180,E1 -1296.748,E2 -1296.748} C_VEL
LIN {X 0,Y 587.31,Z 357.949,A -85,B 0,C 180,E1 -1299.363,E2 -1299.363} C_VEL
LIN {X 0,Y 587.3,Z 357.947,A -85,B 0,C 180,E1 -1302.106,E2 -1302.106} C_VEL
LIN {X 0,Y 587.282,Z 357.959,A -85,B 0,C 180,E1 -1305.087,E2 -1305.087} C_VEL
LIN {X 0,Y 587.295,Z 357.948,A -85,B 0,C 180,E1 -1307.924,E2 -1307.924} C_VEL
LIN {X 0,Y 587.314,Z 357.949,A -85,B 0,C 180,E1 -1310.64,E2 -1310.64} C_VEL
LIN {X 0,Y 587.313,Z 357.952,A -85,B 0,C 180,E1 -1313.298,E2 -1313.298} C_VEL
LIN {X 0,Y 587.319,Z 357.946,A -85,B 0,C 180,E1 -1315.778,E2 -1315.778} C_VEL
LIN {X 0,Y 587.328,Z 357.944,A -85,B 0,C 180,E1 -1318.232,E2 -1318.232} C_VEL
LIN {X 0,Y 587.337,Z 357.95,A -85,B 0,C 180,E1 -1320.87,E2 -1320.87} C_VEL
LIN {X 0,Y 587.306,Z 358.025,A -85,B 0,C 180,E1 -1322.316,E2 -1322.316} C_VEL
LIN {X 0,Y 588.53,Z 362.283,A -85,B 0,C 180,E1 -1322.41,E2 -1322.41} C_VEL
LIN {X 0,Y 588.296,Z 490.55,A -85,B 0,C 180,E1 -1324.03,E2 -1324.03} C_VEL
LIN {X 0,Y 588.226,Z 505.863,A -85,B 0,C 180,E1 -1324.36,E2 -1324.36} C_VEL
LIN {X 0,Y 588.122,Z 520.225,A -85,B 0,C 180,E1 -1324.805,E2 -1324.805} C_VEL
LIN {X 0,Y 587.962,Z 534.652,A -85,B 0,C 180,E1 -1325.393,E2 -1325.393} C_VEL
LIN {X 0,Y 587.804,Z 548.518,A -85,B 0,C 180,E1 -1326.108,E2 -1326.108} C_VEL
LIN {X 0,Y 587.73,Z 561.806,A -85,B 0,C 180,E1 -1326.953,E2 -1326.953} C_VEL
LIN {X 0,Y 587.566,Z 573.779,A -85,B 0,C 180,E1 -1327.867,E2 -1327.867} C_VEL
LIN {X 0,Y 587.459,Z 585.452,A -85,B 0,C 180,E1 -1328.931,E2 -1328.931} C_VEL
LIN {X 0,Y 587.378,Z 595.856,A -85,B 0,C 180,E1 -1330.063,E2 -1330.063} C_VEL
LIN {X 0,Y 587.299,Z 605.6,A -85,B 0,C 180,E1 -1331.331,E2 -1331.331} C_VEL
LIN {X 0,Y 587.248,Z 613.606,A -85,B 0,C 180,E1 -1332.592,E2 -1332.592} C_VEL
LIN {X 0,Y 587.201,Z 621.007,A -85,B 0,C 180,E1 -1334.022,E2 -1334.022} C_VEL
LIN {X 0,Y 587.188,Z 626.778,A -85,B 0,C 180,E1 -1335.443,E2 -1335.443} C_VEL
LIN {X 0,Y 587.143,Z 631.104,A -85,B 0,C 180,E1 -1336.855,E2 -1336.855} C_VEL
LIN {X 0,Y 587.152,Z 634.12,A -85,B 0,C 180,E1 -1338.26,E2 -1338.26} C_VEL
LIN {X 0,Y 587.135,Z 635.9,A -85,B 0,C 180,E1 -1339.657,E2 -1339.657} C_VEL
LIN {X 0,Y 587.121,Z 636.5,A -85,B 0,C 180,E1 -1341.048,E2 -1341.048} C_VEL
LIN {X 0,Y 587.144,Z 635.9,A -85,B 0,C 180,E1 -1342.434,E2 -1342.434} C_VEL
LIN {X 0,Y 587.149,Z 634.144,A -85,B 0,C 180,E1 -1343.816,E2 -1343.816} C_VEL
LIN {X 0,Y 587.131,Z 631.211,A -85,B 0,C 180,E1 -1345.194,E2 -1345.194} C_VEL
LIN {X 0,Y 587.192,Z 627.054,A -85,B 0,C 180,E1 -1346.569,E2 -1346.569} C_VEL
LIN {X 0,Y 587.174,Z 621.594,A -85,B 0,C 180,E1 -1347.943,E2 -1347.943} C_VEL
LIN {X 0,Y 587.241,Z 614.679,A -85,B 0,C 180,E1 -1349.315,E2 -1349.315} C_VEL
LIN {X 0,Y 587.306,Z 606.114,A -85,B 0,C 180,E1 -1350.686,E2 -1350.686} C_VEL
LIN {X 0,Y 587.395,Z 597.057,A -85,B 0,C 180,E1 -1351.886,E2 -1351.886} C_VEL
LIN {X 0,Y 587.443,Z 587.886,A -85,B 0,C 180,E1 -1352.915,E2 -1352.915} C_VEL
LIN {X 0,Y 587.593,Z 577.06,A -85,B 0,C 180,E1 -1353.944,E2 -1353.944} C_VEL
LIN {X 0,Y 587.674,Z 564.156,A -85,B 0,C 180,E1 -1354.974,E2 -1354.974} C_VEL
LIN {X 0,Y 587.844,Z 551.081,A -85,B 0,C 180,E1 -1355.833,E2 -1355.833} C_VEL
LIN {X 0,Y 587.964,Z 537.571,A -85,B 0,C 180,E1 -1356.559,E2 -1356.559} C_VEL
LIN {X 0,Y 588.063,Z 524.113,A -85,B 0,C 180,E1 -1357.141,E2 -1357.141} C_VEL
LIN {X 0,Y 588.174,Z 509.135,A -85,B 0,C 180,E1 -1357.639,E2 -1357.639} C_VEL
LIN {X 0,Y 588.248,Z 494.62,A -85,B 0,C 180,E1 -1357.984,E2 -1357.984} C_VEL
LIN {X 0,Y 588.301,Z 475.533,A -85,B 0,C 180,E1 -1358.264,E2 -1358.264} C_VEL
LIN {X 0,Y 588.406,Z 361.307,A -85,B 0,C 180,E1 -1359.696,E2 -1359.696} C_VEL
LIN {X 0,Y 587.295,Z 357.965,A -85,B 0,C 180,E1 -1359.775,E2 -1359.775} C_VEL
LIN {X 0,Y 587.308,Z 357.948,A -85,B 0,C 180,E1 -1361.738,E2 -1361.738} C_VEL
LIN {X 0,Y 587.299,Z 357.952,A -85,B 0,C 180,E1 -1364.554,E2 -1364.554} C_VEL
LIN {X 0,Y 587.27,Z 357.955,A -85,B 0,C 180,E1 -1367.408,E2 -1367.408} C_VEL
LIN {X 0,Y 587.291,Z 357.951,A -85,B 0,C 180,E1 -1369.577,E2 -1369.577} C_VEL
LIN {X 0,Y 587.266,Z 357.952,A -85,B 0,C 180,E1 -1371.776,E2 -1371.776} C_VEL
LIN {X 0,Y 587.284,Z 357.952,A -85,B 0,C 180,E1 -1374.565,E2 -1374.565} C_VEL
LIN {X 0,Y 587.302,Z 357.958,A -85,B 0,C 180,E1 -1377.047,E2 -1377.047} C_VEL
LIN {X 0,Y 587.288,Z 357.947,A -85,B 0,C 180,E1 -1380.172,E2 -1380.172} C_VEL
LIN {X 0,Y 587.302,Z 357.95,A -85,B 0,C 180,E1 -1382.581,E2 -1382.581} C_VEL
LIN {X 0,Y 587.287,Z 357.958,A -85,B 0,C 180,E1 -1385.058,E2 -1385.058} C_VEL
LIN {X 0,Y 587.306,Z 357.947,A -85,B 0,C 180,E1 -1387.834,E2 -1387.834} C_VEL
LIN {X 0,Y 587.285,Z 357.948,A -85,B 0,C 180,E1 -1390.256,E2 -1390.256} C_VEL
LIN {X 0,Y 587.279,Z 357.96,A -85,B 0,C 180,E1 -1393.114,E2 -1393.114} C_VEL
LIN {X 0,Y 587.29,Z 357.949,A -85,B 0,C 180,E1 -1396.046,E2 -1396.046} C_VEL
LIN {X 0,Y 587.29,Z 357.954,A -85,B 0,C 180,E1 -1398.929,E2 -1398.929} C_VEL
LIN {X 0,Y 587.283,Z 357.955,A -85,B 0,C 180,E1 -1401.517,E2 -1401.517} C_VEL
LIN {X 0,Y 587.266,Z 357.952,A -85,B 0,C 180,E1 -1404.098,E2 -1404.098} C_VEL
LIN {X 0,Y 587.29,Z 357.949,A -85,B 0,C 180,E1 -1406.6,E2 -1406.6} C_VEL
LIN {X 0,Y 587.282,Z 357.955,A -85,B 0,C 180,E1 -1409.03,E2 -1409.03} C_VEL
LIN {X 0,Y 587.287,Z 357.958,A -85,B 0,C 180,E1 -1411.401,E2 -1411.401} C_VEL
LIN {X 0,Y 587.283,Z 357.952,A -85,B 0,C 180,E1 -1413.832,E2 -1413.832} C_VEL
LIN {X 0,Y 587.287,Z 357.95,A -85,B 0,C 180,E1 -1416.74,E2 -1416.74} C_VEL
LIN {X 0,Y 587.301,Z 357.952,A -85,B 0,C 180,E1 -1419.694,E2 -1419.694} C_VEL
LIN {X 0,Y 587.268,Z 357.954,A -85,B 0,C 180,E1 -1421.871,E2 -1421.871} C_VEL
LIN {X 0,Y 587.279,Z 357.951,A -85,B 0,C 180,E1 -1424.023,E2 -1424.023} C_VEL
LIN {X 0,Y 587.311,Z 357.946,A -85,B 0,C 180,E1 -1426.153,E2 -1426.153} C_VEL
LIN {X 0,Y 587.326,Z 357.944,A -85,B 0,C 180,E1 -1428.962,E2 -1428.962} C_VEL
LIN {X 0,Y 587.301,Z 357.952,A -85,B 0,C 180,E1 -1431.744,E2 -1431.744} C_VEL
LIN {X 0,Y 587.281,Z 357.954,A -85,B 0,C 180,E1 -1433.817,E2 -1433.817} C_VEL
LIN {X 0,Y 587.269,Z 357.955,A -85,B 0,C 180,E1 -1435.882,E2 -1435.882} C_VEL
LIN {X 0,Y 587.327,Z 357.947,A -85,B 0,C 180,E1 -1437.943,E2 -1437.943} C_VEL
LIN {X 0,Y 587.343,Z 357.945,A -85,B 0,C 180,E1 -1440,E2 -1440} C_VEL
LIN {X 0,Y 587.323,Z 357.944,A -85,B 0,C 180,E1 -1442.743,E2 -1442.743} C_VEL
LIN {X 0,Y 587.326,Z 357.953,A -85,B 0,C 180,E1 -1445.493,E2 -1445.493} C_VEL
LIN {X 0,Y 587.297,Z 357.948,A -85,B 0,C 180,E1 -1448.256,E2 -1448.256} C_VEL
LIN {X 0,Y 587.319,Z 357.947,A -85,B 0,C 180,E1 -1451.124,E2 -1451.124} C_VEL
LIN {X 0,Y 587.305,Z 357.948,A -85,B 0,C 180,E1 -1454.241,E2 -1454.241} C_VEL
LIN {X 0,Y 587.28,Z 357.95,A -85,B 0,C 180,E1 -1456.796,E2 -1456.796} C_VEL
LIN {X 0,Y 587.285,Z 357.958,A -85,B 0,C 180,E1 -1459.577,E2 -1459.577} C_VEL
LIN {X 0,Y 587.283,Z 357.958,A -85,B 0,C 180,E1 -1461.776,E2 -1461.776} C_VEL
LIN {X 0,Y 587.288,Z 357.949,A -85,B 0,C 180,E1 -1464.761,E2 -1464.761} C_VEL
LIN {X 0,Y 587.287,Z 357.949,A -85,B 0,C 180,E1 -1467.048,E2 -1467.048} C_VEL
LIN {X 0,Y 587.302,Z 357.951,A -85,B 0,C 180,E1 -1470.172,E2 -1470.172} C_VEL
LIN {X 0,Y 587.295,Z 357.948,A -85,B 0,C 180,E1 -1472.582,E2 -1472.582} C_VEL
LIN {X 0,Y 587.285,Z 357.949,A -85,B 0,C 180,E1 -1475.058,E2 -1475.058} C_VEL
LIN {X 0,Y 587.296,Z 357.957,A -85,B 0,C 180,E1 -1477.834,E2 -1477.834} C_VEL
LIN {X 0,Y 587.29,Z 357.952,A -85,B 0,C 180,E1 -1480.256,E2 -1480.256} C_VEL
LIN {X 0,Y 587.27,Z 357.951,A -85,B 0,C 180,E1 -1483.115,E2 -1483.115} C_VEL
LIN {X 0,Y 587.291,Z 357.956,A -85,B 0,C 180,E1 -1486.048,E2 -1486.048} C_VEL
LIN {X 0,Y 587.278,Z 357.948,A -85,B 0,C 180,E1 -1488.931,E2 -1488.931} C_VEL
LIN {X 0,Y 587.304,Z 357.951,A -85,B 0,C 180,E1 -1491.52,E2 -1491.52} C_VEL
LIN {X 0,Y 587.267,Z 357.96,A -85,B 0,C 180,E1 -1494.099,E2 -1494.099} C_VEL
LIN {X 0,Y 587.304,Z 357.949,A -85,B 0,C 180,E1 -1496.602,E2 -1496.602} C_VEL
LIN {X 0,Y 587.31,Z 357.953,A -85,B 0,C 180,E1 -1499.495,E2 -1499.495} C_VEL
LIN {X 0,Y 587.365,Z 358.057,A -85,B 0,C 180,E1 -1499.894,E2 -1499.894} C_VEL
LIN {X 0,Y 588.983,Z 364.451,A -85,B 0,C 180,E1 -1500.583,E2 -1500.583} C_VEL
LIN {X 0,Y 588.787,Z 389.531,A -85,B 0,C 180,E1 -1503.027,E2 -1503.027} C_VEL
LIN {X 0,Y 588.451,Z 419.266,A -85,B 0,C 180,E1 -1505.855,E2 -1505.855} C_VEL
LIN {X 0,Y 588.174,Z 450.326,A -85,B 0,C 180,E1 -1508.75,E2 -1508.75} C_VEL
LIN {X 0,Y 587.96,Z 473.178,A -85,B 0,C 180,E1 -1510.845,E2 -1510.845} C_VEL
LIN {X 0,Y 588.591,Z 478.058,A -85,B 0,C 180,E1 -1510.935,E2 -1510.935} C_VEL
LIN {X 0,Y 588.304,Z 641.283,A -85,B 0,C 180,E1 -1512.998,E2 -1512.998} C_VEL
LIN {X 0,Y 588.211,Z 656.715,A -85,B 0,C 180,E1 -1513.336,E2 -1513.336} C_VEL
LIN {X 0,Y 588.069,Z 672.049,A -85,B 0,C 180,E1 -1513.823,E2 -1513.823} C_VEL
LIN {X 0,Y 587.987,Z 685.767,A -85,B 0,C 180,E1 -1514.399,E2 -1514.399} C_VEL
LIN {X 0,Y 587.828,Z 699.24,A -85,B 0,C 180,E1 -1515.105,E2 -1515.105} C_VEL
LIN {X 0,Y 587.74,Z 712.115,A -85,B 0,C 180,E1 -1515.93,E2 -1515.93} C_VEL
LIN {X 0,Y 587.582,Z 724.288,A -85,B 0,C 180,E1 -1516.864,E2 -1516.864} C_VEL
LIN {X 0,Y 587.453,Z 735.749,A -85,B 0,C 180,E1 -1517.915,E2 -1517.915} C_VEL
LIN {X 0,Y 587.348,Z 745.39,A -85,B 0,C 180,E1 -1518.963,E2 -1518.963} C_VEL
LIN {X 0,Y 587.304,Z 754.856,A -85,B 0,C 180,E1 -1520.182,E2 -1520.182} C_VEL
LIN {X 0,Y 587.264,Z 762.731,A -85,B 0,C 180,E1 -1521.397,E2 -1521.397} C_VEL
LIN {X 0,Y 587.216,Z 770.088,A -85,B 0,C 180,E1 -1522.781,E2 -1522.781} C_VEL
LIN {X 0,Y 587.224,Z 775.924,A -85,B 0,C 180,E1 -1524.161,E2 -1524.161} C_VEL
LIN {X 0,Y 587.136,Z 779.384,A -85,B 0,C 180,E1 -1525.193,E2 -1525.193} C_VEL
LIN {X 0,Y 587.179,Z 782.887,A -85,B 0,C 180,E1 -1526.569,E2 -1526.569} C_VEL
LIN {X 0,Y 587.137,Z 785.193,A -85,B 0,C 180,E1 -1527.942,E2 -1527.942} C_VEL
LIN {X 0,Y 587.137,Z 786.35,A -85,B 0,C 180,E1 -1529.314,E2 -1529.314} C_VEL
LIN {X 0,Y 587.137,Z 786.35,A -85,B 0,C 180,E1 -1530.686,E2 -1530.686} C_VEL
LIN {X 0,Y 587.137,Z 785.193,A -85,B 0,C 180,E1 -1532.058,E2 -1532.058} C_VEL
LIN {X 0,Y 587.179,Z 782.887,A -85,B 0,C 180,E1 -1533.431,E2 -1533.431} C_VEL
LIN {X 0,Y 587.136,Z 779.385,A -85,B 0,C 180,E1 -1534.806,E2 -1534.806} C_VEL
LIN {X 0,Y 587.178,Z 774.61,A -85,B 0,C 180,E1 -1536.184,E2 -1536.184} C_VEL
LIN {X 0,Y 587.235,Z 768.427,A -85,B 0,C 180,E1 -1537.564,E2 -1537.564} C_VEL
LIN {X 0,Y 587.266,Z 760.654,A -85,B 0,C 180,E1 -1538.95,E2 -1538.95} C_VEL
LIN {X 0,Y 587.351,Z 752.374,A -85,B 0,C 180,E1 -1540.165,E2 -1540.165} C_VEL
LIN {X 0,Y 587.399,Z 742.4,A -85,B 0,C 180,E1 -1541.385,E2 -1541.385} C_VEL
LIN {X 0,Y 587.521,Z 732.197,A -85,B 0,C 180,E1 -1542.434,E2 -1542.434} C_VEL
LIN {X 0,Y 587.628,Z 720.025,A -85,B 0,C 180,E1 -1543.486,E2 -1543.486} C_VEL
LIN {X 0,Y 587.773,Z 707.065,A -85,B 0,C 180,E1 -1544.416,E2 -1544.416} C_VEL
LIN {X 0,Y 587.886,Z 692.878,A -85,B 0,C 180,E1 -1545.248,E2 -1545.248} C_VEL
LIN {X 0,Y 588.049,Z 678.812,A -85,B 0,C 180,E1 -1545.91,E2 -1545.91} C_VEL
LIN {X 0,Y 588.168,Z 664.325,A -85,B 0,C 180,E1 -1546.441,E2 -1546.441} C_VEL
LIN {X 0,Y 588.278,Z 649.3,A -85,B 0,C 180,E1 -1546.844,E2 -1546.844} C_VEL
LIN {X 0,Y 588.32,Z 634.113,A -85,B 0,C 180,E1 -1547.109,E2 -1547.109} C_VEL
LIN {X 0,Y 588.541,Z 476.525,A -85,B 0,C 180,E1 -1549.086,E2 -1549.086} C_VEL
LIN {X 0,Y 587.984,Z 473.096,A -85,B 0,C 180,E1 -1549.161,E2 -1549.161} C_VEL
LIN {X 0,Y 588.228,Z 443.059,A -85,B 0,C 180,E1 -1551.923,E2 -1551.923} C_VEL
LIN {X 0,Y 588.522,Z 413.325,A -85,B 0,C 180,E1 -1554.705,E2 -1554.705} C_VEL
LIN {X 0,Y 588.842,Z 383.591,A -85,B 0,C 180,E1 -1557.547,E2 -1557.547} C_VEL
LIN {X 0,Y 588.917,Z 363.772,A -85,B 0,C 180,E1 -1559.488,E2 -1559.488} C_VEL
LIN {X 0,Y 587.354,Z 357.95,A -85,B 0,C 180,E1 -1560.118,E2 -1560.118} C_VEL
LIN {X 0,Y 587.325,Z 357.945,A -85,B 0,C 180,E1 -1563.11,E2 -1563.11} C_VEL
LIN {X 0,Y 587.265,Z 357.96,A -85,B 0,C 180,E1 -1565.901,E2 -1565.901} C_VEL
LIN {X 0,Y 587.303,Z 357.952,A -85,B 0,C 180,E1 -1568.48,E2 -1568.48} C_VEL
LIN {X 0,Y 587.292,Z 357.948,A -85,B 0,C 180,E1 -1571.159,E2 -1571.159} C_VEL
LIN {X 0,Y 587.287,Z 357.956,A -85,B 0,C 180,E1 -1573.952,E2 -1573.952} C_VEL
LIN {X 0,Y 587.262,Z 357.952,A -85,B 0,C 180,E1 -1576.989,E2 -1576.989} C_VEL
LIN {X 0,Y 587.287,Z 357.952,A -85,B 0,C 180,E1 -1579.743,E2 -1579.743} C_VEL
LIN {X 0,Y 587.298,Z 357.955,A -85,B 0,C 180,E1 -1582.389,E2 -1582.389} C_VEL
LIN {X 0,Y 587.308,Z 357.948,A -85,B 0,C 180,E1 -1585.655,E2 -1585.655} C_VEL
LIN {X 0,Y 587.317,Z 357.955,A -85,B 0,C 180,E1 -1588.23,E2 -1588.23} C_VEL
LIN {X 0,Y 587.282,Z 357.952,A -85,B 0,C 180,E1 -1590.875,E2 -1590.875} C_VEL
LIN {X 0,Y 587.292,Z 357.951,A -85,B 0,C 180,E1 -1593.829,E2 -1593.829} C_VEL
LIN {X 0,Y 587.273,Z 357.955,A -85,B 0,C 180,E1 -1596.739,E2 -1596.739} C_VEL
LIN {X 0,Y 587.282,Z 357.95,A -85,B 0,C 180,E1 -1599.694,E2 -1599.694} C_VEL
LIN {X 0,Y 587.256,Z 357.955,A -85,B 0,C 180,E1 -1601.871,E2 -1601.871} C_VEL
LIN {X 0,Y 587.282,Z 357.955,A -85,B 0,C 180,E1 -1604.736,E2 -1604.736} C_VEL
LIN {X 0,Y 587.255,Z 357.957,A -85,B 0,C 180,E1 -1606.857,E2 -1606.857} C_VEL
LIN {X 0,Y 587.32,Z 357.947,A -85,B 0,C 180,E1 -1608.962,E2 -1608.962} C_VEL
LIN {X 0,Y 587.296,Z 357.948,A -85,B 0,C 180,E1 -1611.744,E2 -1611.744} C_VEL
LIN {X 0,Y 587.329,Z 357.954,A -85,B 0,C 180,E1 -1614.507,E2 -1614.507} C_VEL
LIN {X 0,Y 587.324,Z 357.944,A -85,B 0,C 180,E1 -1617.257,E2 -1617.257} C_VEL
LIN {X 0,Y 587.341,Z 357.944,A -85,B 0,C 180,E1 -1620,E2 -1620} C_VEL
LIN {X 0,Y 587.358,Z 357.948,A -85,B 0,C 180,E1 -1622.744,E2 -1622.744} C_VEL
LIN {X 0,Y 587.307,Z 357.945,A -85,B 0,C 180,E1 -1625.494,E2 -1625.494} C_VEL
LIN {X 0,Y 587.287,Z 357.946,A -85,B 0,C 180,E1 -1627.564,E2 -1627.564} C_VEL
LIN {X 0,Y 587.267,Z 357.951,A -85,B 0,C 180,E1 -1629.645,E2 -1629.645} C_VEL
LIN {X 0,Y 587.302,Z 357.947,A -85,B 0,C 180,E1 -1631.738,E2 -1631.738} C_VEL
LIN {X 0,Y 587.316,Z 357.951,A -85,B 0,C 180,E1 -1634.554,E2 -1634.554} C_VEL
LIN {X 0,Y 587.293,Z 357.949,A -85,B 0,C 180,E1 -1637.408,E2 -1637.408} C_VEL
LIN {X 0,Y 587.281,Z 357.952,A -85,B 0,C 180,E1 -1638.325,E2 -1638.325} C_VEL
LIN {X 0,Y 586.651,Z 358.036,A -85,B 0,C 180,E1 -1638.897,E2 -1638.897} C_VEL
LIN {X 0,Y 583.836,Z 358.386,A -85,B 0,C 180,E1 -1639.826,E2 -1639.826} C_VEL
LIN {X 0,Y 581.423,Z 358.685,A -85,B 0,C 180,E1 -1640.573,E2 -1640.573} C_VEL
LIN {X 0,Y 580.362,Z 358.815,A -85,B 0,C 180,E1 -1641.149,E2 -1641.149} C_VEL
LIN {X 0,Y 580.264,Z 358.824,A -85,B 0,C 180,E1 -1641.345,E2 -1641.345} C_VEL
LIN {X 0,Y 580.243,Z 358.827,A -85,B 0,C 180,E1 -1643.56,E2 -1643.56} C_VEL
LIN {X 0,Y 580.239,Z 358.829,A -85,B 0,C 180,E1 -1646.327,E2 -1646.327} C_VEL
LIN {X 0,Y 580.265,Z 358.827,A -85,B 0,C 180,E1 -1649.306,E2 -1649.306} C_VEL
LIN {X 0,Y 580.283,Z 358.821,A -85,B 0,C 180,E1 -1652.202,E2 -1652.202} C_VEL
LIN {X 0,Y 580.276,Z 358.83,A -85,B 0,C 180,E1 -1654.698,E2 -1654.698} C_VEL
LIN {X 0,Y 580.283,Z 358.826,A -85,B 0,C 180,E1 -1657.27,E2 -1657.27} C_VEL
LIN {X 0,Y 580.273,Z 358.823,A -85,B 0,C 180,E1 -1660.27,E2 -1660.27} C_VEL
LIN {X 0,Y 580.256,Z 358.831,A -85,B 0,C 180,E1 -1662.709,E2 -1662.709} C_VEL
LIN {X 0,Y 580.247,Z 358.828,A -85,B 0,C 180,E1 -1665.612,E2 -1665.612} C_VEL
LIN {X 0,Y 580.265,Z 358.829,A -85,B 0,C 180,E1 -1668.671,E2 -1668.671} C_VEL
LIN {X 0,Y 580.262,Z 358.833,A -85,B 0,C 180,E1 -1670.965,E2 -1670.965} C_VEL
LIN {X 0,Y 580.24,Z 358.829,A -85,B 0,C 180,E1 -1673.596,E2 -1673.596} C_VEL
LIN {X 0,Y 580.269,Z 358.824,A -85,B 0,C 180,E1 -1676.143,E2 -1676.143} C_VEL
LIN {X 0,Y 580.262,Z 358.827,A -85,B 0,C 180,E1 -1678.615,E2 -1678.615} C_VEL
LIN {X 0,Y 580.276,Z 358.832,A -85,B 0,C 180,E1 -1681.024,E2 -1681.024} C_VEL
LIN {X 0,Y 580.262,Z 358.827,A -85,B 0,C 180,E1 -1682.081,E2 -1682.081} C_VEL
LIN {X 0,Y 581.83,Z 363.697,A -85,B 0,C 180,E1 -1682.206,E2 -1682.206} C_VEL
LIN {X 0,Y 581.521,Z 490.511,A -85,B 0,C 180,E1 -1683.826,E2 -1683.826} C_VEL
LIN {X 0,Y 581.434,Z 505.838,A -85,B 0,C 180,E1 -1684.158,E2 -1684.158} C_VEL
LIN {X 0,Y 581.277,Z 520.876,A -85,B 0,C 180,E1 -1684.631,E2 -1684.631} C_VEL
LIN {X 0,Y 581.089,Z 535.503,A -85,B 0,C 180,E1 -1685.242,E2 -1685.242} C_VEL
LIN {X 0,Y 580.916,Z 549.74,A -85,B 0,C 180,E1 -1685.997,E2 -1685.997} C_VEL
LIN {X 0,Y 580.792,Z 563.174,A -85,B 0,C 180,E1 -1686.876,E2 -1686.876} C_VEL
LIN {X 0,Y 580.597,Z 575.71,A -85,B 0,C 180,E1 -1687.868,E2 -1687.868} C_VEL
LIN {X 0,Y 580.446,Z 587.551,A -85,B 0,C 180,E1 -1688.994,E2 -1688.994} C_VEL
LIN {X 0,Y 580.304,Z 597.942,A -85,B 0,C 180,E1 -1690.178,E2 -1690.178} C_VEL
LIN {X 0,Y 580.256,Z 607.318,A -85,B 0,C 180,E1 -1691.463,E2 -1691.463} C_VEL
LIN {X 0,Y 580.184,Z 615.034,A -85,B 0,C 180,E1 -1692.737,E2 -1692.737} C_VEL
LIN {X 0,Y 580.128,Z 622.142,A -85,B 0,C 180,E1 -1694.183,E2 -1694.183} C_VEL
LIN {X 0,Y 580.124,Z 626.379,A -85,B 0,C 180,E1 -1695.262,E2 -1695.262} C_VEL
LIN {X 0,Y 580.063,Z 630.818,A -85,B 0,C 180,E1 -1696.692,E2 -1696.692} C_VEL
LIN {X 0,Y 580.051,Z 633.939,A -85,B 0,C 180,E1 -1698.114,E2 -1698.114} C_VEL
LIN {X 0,Y 580.055,Z 635.821,A -85,B 0,C 180,E1 -1699.529,E2 -1699.529} C_VEL
LIN {X 0,Y 580.02,Z 636.482,A -85,B 0,C 180,E1 -1700.938,E2 -1700.938} C_VEL
LIN {X 0,Y 580.065,Z 635.975,A -85,B 0,C 180,E1 -1702.342,E2 -1702.342} C_VEL
LIN {X 0,Y 580.067,Z 634.319,A -85,B 0,C 180,E1 -1703.74,E2 -1703.74} C_VEL
LIN {X 0,Y 580.034,Z 631.492,A -85,B 0,C 180,E1 -1705.135,E2 -1705.135} C_VEL
LIN {X 0,Y 580.121,Z 627.442,A -85,B 0,C 180,E1 -1706.528,E2 -1706.528} C_VEL
LIN {X 0,Y 580.085,Z 622.098,A -85,B 0,C 180,E1 -1707.917,E2 -1707.917} C_VEL
LIN {X 0,Y 580.174,Z 615.298,A -85,B 0,C 180,E1 -1709.306,E2 -1709.306} C_VEL
LIN {X 0,Y 580.256,Z 606.88,A -85,B 0,C 180,E1 -1710.694,E2 -1710.694} C_VEL
LIN {X 0,Y 580.342,Z 597.958,A -85,B 0,C 180,E1 -1711.909,E2 -1711.909} C_VEL
LIN {X 0,Y 580.457,Z 587.289,A -85,B 0,C 180,E1 -1713.123,E2 -1713.123} C_VEL
LIN {X 0,Y 580.611,Z 575.351,A -85,B 0,C 180,E1 -1714.252,E2 -1714.252} C_VEL
LIN {X 0,Y 580.759,Z 563.27,A -85,B 0,C 180,E1 -1715.207,E2 -1715.207} C_VEL
LIN {X 0,Y 580.968,Z 550.01,A -85,B 0,C 180,E1 -1716.076,E2 -1716.076} C_VEL
LIN {X 0,Y 581.127,Z 537.074,A -85,B 0,C 180,E1 -1716.772,E2 -1716.772} C_VEL
LIN {X 0,Y 581.247,Z 522.308,A -85,B 0,C 180,E1 -1717.407,E2 -1717.407} C_VEL
LIN {X 0,Y 581.385,Z 506.939,A -85,B 0,C 180,E1 -1717.904,E2 -1717.904} C_VEL
LIN {X 0,Y 581.479,Z 491.329,A -85,B 0,C 180,E1 -1718.252,E2 -1718.252} C_VEL
LIN {X 0,Y 581.805,Z 363.304,A -85,B 0,C 180,E1 -1719.89,E2 -1719.89} C_VEL
LIN {X 0,Y 580.249,Z 358.829,A -85,B 0,C 180,E1 -1720.005,E2 -1720.005} C_VEL
LIN {X 0,Y 580.279,Z 358.824,A -85,B 0,C 180,E1 -1721.882,E2 -1721.882} C_VEL
LIN {X 0,Y 580.259,Z 358.832,A -85,B 0,C 180,E1 -1724.735,E2 -1724.735} C_VEL
LIN {X 0,Y 580.235,Z 358.829,A -85,B 0,C 180,E1 -1727.626,E2 -1727.626} C_VEL
LIN {X 0,Y 580.251,Z 358.826,A -85,B 0,C 180,E1 -1729.824,E2 -1729.824} C_VEL
LIN {X 0,Y 580.21,Z 358.831,A -85,B 0,C 180,E1 -1732.055,E2 -1732.055} C_VEL
LIN {X 0,Y 580.239,Z 358.832,A -85,B 0,C 180,E1 -1734.712,E2 -1734.712} C_VEL
LIN {X 0,Y 580.244,Z 358.831,A -85,B 0,C 180,E1 -1737.403,E2 -1737.403} C_VEL
LIN {X 0,Y 580.242,Z 358.825,A -85,B 0,C 180,E1 -1739.775,E2 -1739.775} C_VEL
LIN {X 0,Y 580.266,Z 358.824,A -85,B 0,C 180,E1 -1742.202,E2 -1742.202} C_VEL
LIN {X 0,Y 580.266,Z 358.827,A -85,B 0,C 180,E1 -1744.697,E2 -1744.697} C_VEL
LIN {X 0,Y 580.275,Z 358.831,A -85,B 0,C 180,E1 -1747.269,E2 -1747.269} C_VEL
LIN {X 0,Y 580.266,Z 358.823,A -85,B 0,C 180,E1 -1750.267,E2 -1750.267} C_VEL
LIN {X 0,Y 580.239,Z 358.83,A -85,B 0,C 180,E1 -1752.709,E2 -1752.709} C_VEL
LIN {X 0,Y 580.241,Z 358.83,A -85,B 0,C 180,E1 -1755.611,E2 -1755.611} C_VEL
LIN {X 0,Y 580.228,Z 358.828,A -85,B 0,C 180,E1 -1758.226,E2 -1758.226} C_VEL
LIN {X 0,Y 580.247,Z 358.832,A -85,B 0,C 180,E1 -1760.962,E2 -1760.962} C_VEL
LIN {X 0,Y 580.232,Z 358.833,A -85,B 0,C 180,E1 -1763.593,E2 -1763.593} C_VEL
LIN {X 0,Y 580.255,Z 358.824,A -85,B 0,C 180,E1 -1766.141,E2 -1766.141} C_VEL
LIN {X 0,Y 580.236,Z 358.828,A -85,B 0,C 180,E1 -1768.612,E2 -1768.612} C_VEL
LIN {X 0,Y 580.257,Z 358.83,A -85,B 0,C 180,E1 -1771.022,E2 -1771.022} C_VEL
LIN {X 0,Y 580.237,Z 358.832,A -85,B 0,C 180,E1 -1773.675,E2 -1773.675} C_VEL
LIN {X 0,Y 580.239,Z 358.826,A -85,B 0,C 180,E1 -1776.44,E2 -1776.44} C_VEL
LIN {X 0,Y 580.253,Z 358.834,A -85,B 0,C 180,E1 -1779.436,E2 -1779.436} C_VEL
LIN {X 0,Y 580.23,Z 358.834,A -85,B 0,C 180,E1 -1781.644,E2 -1781.644} C_VEL
LIN {X 0,Y 580.259,Z 358.824,A -85,B 0,C 180,E1 -1784.546,E2 -1784.546} C_VEL
LIN {X 0,Y 580.274,Z 358.83,A -85,B 0,C 180,E1 -1787.408,E2 -1787.408} C_VEL
LIN {X 0,Y 580.25,Z 358.831,A -85,B 0,C 180,E1 -1789.532,E2 -1789.532} C_VEL
LIN {X 0,Y 580.239,Z 358.826,A -85,B 0,C 180,E1 -1792.343,E2 -1792.343} C_VEL
LIN {X 0,Y 580.272,Z 358.823,A -85,B 0,C 180,E1 -1794.44,E2 -1794.44} C_VEL
LIN {X 0,Y 580.316,Z 358.822,A -85,B 0,C 180,E1 -1797.223,E2 -1797.223} C_VEL
LIN {X 0,Y 580.314,Z 358.82,A -85,B 0,C 180,E1 -1800,E2 -1800} C_VEL
LIN {X 0,Y 580.294,Z 358.82,A -85,B 0,C 180,E1 -1802.777,E2 -1802.777} C_VEL
LIN {X 0,Y 580.291,Z 358.83,A -85,B 0,C 180,E1 -1805.56,E2 -1805.56} C_VEL
LIN {X 0,Y 580.268,Z 358.823,A -85,B 0,C 180,E1 -1808.357,E2 -1808.357} C_VEL
LIN {X 0,Y 580.29,Z 358.824,A -85,B 0,C 180,E1 -1811.191,E2 -1811.191} C_VEL
LIN {X 0,Y 580.267,Z 358.823,A -85,B 0,C 180,E1 -1814.324,E2 -1814.324} C_VEL
LIN {X 0,Y 580.238,Z 358.828,A -85,B 0,C 180,E1 -1816.899,E2 -1816.899} C_VEL
LIN {X 0,Y 580.258,Z 358.833,A -85,B 0,C 180,E1 -1819.824,E2 -1819.824} C_VEL
LIN {X 0,Y 580.218,Z 358.833,A -85,B 0,C 180,E1 -1822.055,E2 -1822.055} C_VEL
LIN {X 0,Y 580.269,Z 358.824,A -85,B 0,C 180,E1 -1825.081,E2 -1825.081} C_VEL
LIN {X 0,Y 580.228,Z 358.837,A -85,B 0,C 180,E1 -1827.848,E2 -1827.848} C_VEL
LIN {X 0,Y 580.255,Z 358.825,A -85,B 0,C 180,E1 -1830.691,E2 -1830.691} C_VEL
LIN {X 0,Y 580.258,Z 358.827,A -85,B 0,C 180,E1 -1833.311,E2 -1833.311} C_VEL
LIN {X 0,Y 580.216,Z 358.839,A -85,B 0,C 180,E1 -1835.754,E2 -1835.754} C_VEL
LIN {X 0,Y 580.257,Z 358.828,A -85,B 0,C 180,E1 -1838.149,E2 -1838.149} C_VEL
LIN {X 0,Y 580.265,Z 358.824,A -85,B 0,C 180,E1 -1840.846,E2 -1840.846} C_VEL
LIN {X 0,Y 580.217,Z 358.836,A -85,B 0,C 180,E1 -1843.664,E2 -1843.664} C_VEL
LIN {X 0,Y 580.225,Z 358.83,A -85,B 0,C 180,E1 -1846.615,E2 -1846.615} C_VEL
LIN {X 0,Y 580.232,Z 358.827,A -85,B 0,C 180,E1 -1849.152,E2 -1849.152} C_VEL
LIN {X 0,Y 580.272,Z 358.833,A -85,B 0,C 180,E1 -1851.929,E2 -1851.929} C_VEL
LIN {X 0,Y 580.213,Z 358.834,A -85,B 0,C 180,E1 -1854.451,E2 -1854.451} C_VEL
LIN {X 0,Y 580.239,Z 358.829,A -85,B 0,C 180,E1 -1856.972,E2 -1856.972} C_VEL
LIN {X 0,Y 580.297,Z 358.948,A -85,B 0,C 180,E1 -1859.665,E2 -1859.665} C_VEL
LIN {X 0,Y 582.092,Z 365.605,A -85,B 0,C 180,E1 -1860.378,E2 -1860.378} C_VEL
LIN {X 0,Y 582.301,Z 376.621,A -85,B 0,C 180,E1 -1861.43,E2 -1861.43} C_VEL
LIN {X 0,Y 581.906,Z 405.39,A -85,B 0,C 180,E1 -1864.228,E2 -1864.228} C_VEL
LIN {X 0,Y 581.539,Z 434.507,A -85,B 0,C 180,E1 -1867.003,E2 -1867.003} C_VEL
LIN {X 0,Y 581.237,Z 462.876,A -85,B 0,C 180,E1 -1869.658,E2 -1869.658} C_VEL
LIN {X 0,Y 581.114,Z 473.274,A -85,B 0,C 180,E1 -1870.619,E2 -1870.619} C_VEL
LIN {X 0,Y 581.888,Z 479.174,A -85,B 0,C 180,E1 -1870.721,E2 -1870.721} C_VEL
LIN {X 0,Y 581.531,Z 641.449,A -85,B 0,C 180,E1 -1872.797,E2 -1872.797} C_VEL
LIN {X 0,Y 581.414,Z 656.714,A -85,B 0,C 180,E1 -1873.136,E2 -1873.136} C_VEL
LIN {X 0,Y 581.244,Z 672.048,A -85,B 0,C 180,E1 -1873.628,E2 -1873.628} C_VEL
LIN {X 0,Y 581.123,Z 685.77,A -85,B 0,C 180,E1 -1874.21,E2 -1874.21} C_VEL
LIN {X 0,Y 580.943,Z 699.242,A -85,B 0,C 180,E1 -1874.924,E2 -1874.924} C_VEL
LIN {X 0,Y 580.804,Z 712.48,A -85,B 0,C 180,E1 -1875.783,E2 -1875.783} C_VEL
LIN {X 0,Y 580.608,Z 724.289,A -85,B 0,C 180,E1 -1876.704,E2 -1876.704} C_VEL
LIN {X 0,Y 580.479,Z 735.749,A -85,B 0,C 180,E1 -1877.768,E2 -1877.768} C_VEL
LIN {X 0,Y 580.307,Z 746.454,A -85,B 0,C 180,E1 -1878.953,E2 -1878.953} C_VEL
LIN {X 0,Y 580.268,Z 754.857,A -85,B 0,C 180,E1 -1880.061,E2 -1880.061} C_VEL
LIN {X 0,Y 580.214,Z 762.732,A -85,B 0,C 180,E1 -1881.291,E2 -1881.291} C_VEL
LIN {X 0,Y 580.131,Z 770.088,A -85,B 0,C 180,E1 -1882.692,E2 -1882.692} C_VEL
LIN {X 0,Y 580.129,Z 775.923,A -85,B 0,C 180,E1 -1884.089,E2 -1884.089} C_VEL
LIN {X 0,Y 580.041,Z 779.384,A -85,B 0,C 180,E1 -1885.134,E2 -1885.134} C_VEL
LIN {X 0,Y 580.105,Z 782.888,A -85,B 0,C 180,E1 -1886.527,E2 -1886.527} C_VEL
LIN {X 0,Y 580.036,Z 785.193,A -85,B 0,C 180,E1 -1887.917,E2 -1887.917} C_VEL
LIN {X 0,Y 580.038,Z 786.349,A -85,B 0,C 180,E1 -1889.306,E2 -1889.306} C_VEL
LIN {X 0,Y 580.038,Z 786.349,A -85,B 0,C 180,E1 -1890.694,E2 -1890.694} C_VEL
LIN {X 0,Y 580.036,Z 785.192,A -85,B 0,C 180,E1 -1892.083,E2 -1892.083} C_VEL
LIN {X 0,Y 580.105,Z 782.887,A -85,B 0,C 180,E1 -1893.472,E2 -1893.472} C_VEL
LIN {X 0,Y 580.041,Z 779.386,A -85,B 0,C 180,E1 -1894.865,E2 -1894.865} C_VEL
LIN {X 0,Y 580.091,Z 774.61,A -85,B 0,C 180,E1 -1896.259,E2 -1896.259} C_VEL
LIN {X 0,Y 580.168,Z 768.426,A -85,B 0,C 180,E1 -1897.657,E2 -1897.657} C_VEL
LIN {X 0,Y 580.207,Z 760.653,A -85,B 0,C 180,E1 -1899.059,E2 -1899.059} C_VEL
LIN {X 0,Y 580.308,Z 752.373,A -85,B 0,C 180,E1 -1900.29,E2 -1900.29} C_VEL
LIN {X 0,Y 580.382,Z 742.4,A -85,B 0,C 180,E1 -1901.525,E2 -1901.525} C_VEL
LIN {X 0,Y 580.54,Z 732.196,A -85,B 0,C 180,E1 -1902.586,E2 -1902.586} C_VEL
LIN {X 0,Y 580.677,Z 720.026,A -85,B 0,C 180,E1 -1903.651,E2 -1903.651} C_VEL
LIN {X 0,Y 580.844,Z 707.815,A -85,B 0,C 180,E1 -1904.541,E2 -1904.541} C_VEL
LIN {X 0,Y 580.985,Z 694.531,A -85,B 0,C 180,E1 -1905.343,E2 -1905.343} C_VEL
LIN {X 0,Y 581.201,Z 679.851,A -85,B 0,C 180,E1 -1906.057,E2 -1906.057} C_VEL
LIN {X 0,Y 581.34,Z 665.637,A -85,B 0,C 180,E1 -1906.595,E2 -1906.595} C_VEL
LIN {X 0,Y 581.471,Z 651.192,A -85,B 0,C 180,E1 -1907,E2 -1907} C_VEL
LIN {X 0,Y 581.518,Z 636.859,A -85,B 0,C 180,E1 -1907.275,E2 -1907.275} C_VEL
LIN {X 0,Y 581.897,Z 478.452,A -85,B 0,C 180,E1 -1909.288,E2 -1909.288} C_VEL
LIN {X 0,Y 581.115,Z 473.262,A -85,B 0,C 180,E1 -1909.382,E2 -1909.382} C_VEL
LIN {X 0,Y 581.439,Z 443.059,A -85,B 0,C 180,E1 -1912.192,E2 -1912.192} C_VEL
LIN {X 0,Y 581.816,Z 412.924,A -85,B 0,C 180,E1 -1915.048,E2 -1915.048} C_VEL
LIN {X 0,Y 582.227,Z 383.591,A -85,B 0,C 180,E1 -1917.887,E2 -1917.887} C_VEL
LIN {X 0,Y 582.27,Z 367.302,A -85,B 0,C 180,E1 -1919.449,E2 -1919.449} C_VEL
LIN {X 0,Y 581.787,Z 364.302,A -85,B 0,C 180,E1 -1919.752,E2 -1919.752} C_VEL
LIN {X 0,Y 580.286,Z 358.831,A -85,B 0,C 180,E1 -1920.348,E2 -1920.348} C_VEL
LIN {X 0,Y 580.272,Z 358.825,A -85,B 0,C 180,E1 -1923.312,E2 -1923.312} C_VEL
LIN {X 0,Y 580.213,Z 358.836,A -85,B 0,C 180,E1 -1925.752,E2 -1925.752} C_VEL
LIN {X 0,Y 580.268,Z 358.833,A -85,B 0,C 180,E1 -1928.146,E2 -1928.146} C_VEL
LIN {X 0,Y 580.263,Z 358.825,A -85,B 0,C 180,E1 -1930.845,E2 -1930.845} C_VEL
LIN {X 0,Y 580.222,Z 358.83,A -85,B 0,C 180,E1 -1933.385,E2 -1933.385} C_VEL
LIN {X 0,Y 580.214,Z 358.838,A -85,B 0,C 180,E1 -1936.336,E2 -1936.336} C_VEL
LIN {X 0,Y 580.262,Z 358.824,A -85,B 0,C 180,E1 -1939.154,E2 -1939.154} C_VEL
LIN {X 0,Y 580.259,Z 358.829,A -85,B 0,C 180,E1 -1941.929,E2 -1941.929} C_VEL
LIN {X 0,Y 580.212,Z 358.838,A -85,B 0,C 180,E1 -1944.45,E2 -1944.45} C_VEL
LIN {X 0,Y 580.225,Z 358.83,A -85,B 0,C 180,E1 -1946.971,E2 -1946.971} C_VEL
LIN {X 0,Y 580.261,Z 358.824,A -85,B 0,C 180,E1 -1949.423,E2 -1949.423} C_VEL
LIN {X 0,Y 580.221,Z 358.837,A -85,B 0,C 180,E1 -1952.152,E2 -1952.152} C_VEL
LIN {X 0,Y 580.266,Z 358.825,A -85,B 0,C 180,E1 -1954.919,E2 -1954.919} C_VEL
LIN {X 0,Y 580.213,Z 358.834,A -85,B 0,C 180,E1 -1957.945,E2 -1957.945} C_VEL
LIN {X 0,Y 580.258,Z 358.827,A -85,B 0,C 180,E1 -1960.912,E2 -1960.912} C_VEL
LIN {X 0,Y 580.218,Z 358.831,A -85,B 0,C 180,E1 -1963.824,E2 -1963.824} C_VEL
LIN {X 0,Y 580.262,Z 358.827,A -85,B 0,C 180,E1 -1965.982,E2 -1965.982} C_VEL
LIN {X 0,Y 580.289,Z 358.825,A -85,B 0,C 180,E1 -1968.827,E2 -1968.827} C_VEL
LIN {X 0,Y 580.269,Z 358.823,A -85,B 0,C 180,E1 -1971.643,E2 -1971.643} C_VEL
LIN {X 0,Y 580.293,Z 358.829,A -85,B 0,C 180,E1 -1974.44,E2 -1974.44} C_VEL
LIN {X 0,Y 580.294,Z 358.82,A -85,B 0,C 180,E1 -1977.223,E2 -1977.223} C_VEL
LIN {X 0,Y 580.311,Z 358.82,A -85,B 0,C 180,E1 -1980,E2 -1980} C_VEL
LIN {X 0,Y 580.32,Z 358.824,A -85,B 0,C 180,E1 -1982.777,E2 -1982.777} C_VEL
LIN {X 0,Y 580.275,Z 358.82,A -85,B 0,C 180,E1 -1985.56,E2 -1985.56} C_VEL
LIN {X 0,Y 580.24,Z 358.823,A -85,B 0,C 180,E1 -1987.657,E2 -1987.657} C_VEL
LIN {X 0,Y 580.257,Z 358.831,A -85,B 0,C 180,E1 -1990.468,E2 -1990.468} C_VEL
LIN {X 0,Y 580.277,Z 358.831,A -85,B 0,C 180,E1 -1992.592,E2 -1992.592} C_VEL
LIN {X 0,Y 580.265,Z 358.823,A -85,B 0,C 180,E1 -1995.454,E2 -1995.454} C_VEL
LIN {X 0,Y 580.248,Z 358.826,A -85,B 0,C 180,E1 -1997.626,E2 -1997.626} C_VEL
LIN {X 0,Y 580.265,Z 358.822,A -85,B 0,C 180,E1 -1999.824,E2 -1999.824} C_VEL
LIN {X 0,Y 580.264,Z 358.824,A -85,B 0,C 180,E1 -2001.345,E2 -2001.345} C_VEL
LIN {X 0,Y 579.559,Z 358.913,A -85,B 0,C 180,E1 -2001.924,E2 -2001.924} C_VEL
LIN {X 0,Y 576.677,Z 359.28,A -85,B 0,C 180,E1 -2002.863,E2 -2002.863} C_VEL
LIN {X 0,Y 574.276,Z 359.574,A -85,B 0,C 180,E1 -2003.62,E2 -2003.62} C_VEL
LIN {X 0,Y 573.265,Z 359.698,A -85,B 0,C 180,E1 -2004.203,E2 -2004.203} C_VEL
LIN {X 0,Y 573.193,Z 359.709,A -85,B 0,C 180,E1 -2004.401,E2 -2004.401} C_VEL
LIN {X 0,Y 573.174,Z 359.714,A -85,B 0,C 180,E1 -2006.98,E2 -2006.98} C_VEL
LIN {X 0,Y 573.211,Z 359.704,A -85,B 0,C 180,E1 -2009.485,E2 -2009.485} C_VEL
LIN {X 0,Y 573.236,Z 359.699,A -85,B 0,C 180,E1 -2012.228,E2 -2012.228} C_VEL
LIN {X 0,Y 573.223,Z 359.71,A -85,B 0,C 180,E1 -2014.772,E2 -2014.772} C_VEL
LIN {X 0,Y 573.219,Z 359.702,A -85,B 0,C 180,E1 -2017.809,E2 -2017.809} C_VEL
LIN {X 0,Y 573.236,Z 359.703,A -85,B 0,C 180,E1 -2020.526,E2 -2020.526} C_VEL
LIN {X 0,Y 573.199,Z 359.707,A -85,B 0,C 180,E1 -2023.363,E2 -2023.363} C_VEL
LIN {X 0,Y 573.228,Z 359.702,A -85,B 0,C 180,E1 -2026.333,E2 -2026.333} C_VEL
LIN {X 0,Y 573.239,Z 359.702,A -85,B 0,C 180,E1 -2029.476,E2 -2029.476} C_VEL
LIN {X 0,Y 573.221,Z 359.701,A -85,B 0,C 180,E1 -2032.193,E2 -2032.193} C_VEL
LIN {X 0,Y 573.22,Z 359.71,A -85,B 0,C 180,E1 -2035.231,E2 -2035.231} C_VEL
LIN {X 0,Y 573.234,Z 359.701,A -85,B 0,C 180,E1 -2037.775,E2 -2037.775} C_VEL
LIN {X 0,Y 573.23,Z 359.705,A -85,B 0,C 180,E1 -2040.633,E2 -2040.633} C_VEL
LIN {X 0,Y 573.221,Z 359.808,A -85,B 0,C 180,E1 -2041.861,E2 -2041.861} C_VEL
LIN {X 0,Y 575.058,Z 364.894,A -85,B 0,C 180,E1 -2041.991,E2 -2041.991} C_VEL
LIN {X 0,Y 574.739,Z 490.388,A -85,B 0,C 180,E1 -2043.614,E2 -2043.614} C_VEL
LIN {X 0,Y 574.645,Z 505.808,A -85,B 0,C 180,E1 -2043.952,E2 -2043.952} C_VEL
LIN {X 0,Y 574.455,Z 520.161,A -85,B 0,C 180,E1 -2044.405,E2 -2044.405} C_VEL
LIN {X 0,Y 574.272,Z 534.663,A -85,B 0,C 180,E1 -2045.011,E2 -2045.011} C_VEL
LIN {X 0,Y 574.044,Z 547.653,A -85,B 0,C 180,E1 -2045.691,E2 -2045.691} C_VEL
LIN {X 0,Y 573.836,Z 561.401,A -85,B 0,C 180,E1 -2046.575,E2 -2046.575} C_VEL
LIN {X 0,Y 573.65,Z 574.302,A -85,B 0,C 180,E1 -2047.585,E2 -2047.585} C_VEL
LIN {X 0,Y 573.474,Z 585.673,A -85,B 0,C 180,E1 -2048.653,E2 -2048.653} C_VEL
LIN {X 0,Y 573.358,Z 595.443,A -85,B 0,C 180,E1 -2049.741,E2 -2049.741} C_VEL
LIN {X 0,Y 573.183,Z 605.368,A -85,B 0,C 180,E1 -2051.057,E2 -2051.057} C_VEL
LIN {X 0,Y 573.107,Z 613.327,A -85,B 0,C 180,E1 -2052.332,E2 -2052.332} C_VEL
LIN {X 0,Y 573.041,Z 619.952,A -85,B 0,C 180,E1 -2053.616,E2 -2053.616} C_VEL
LIN {X 0,Y 573.028,Z 625.975,A -85,B 0,C 180,E1 -2055.075,E2 -2055.075} C_VEL
LIN {X 0,Y 572.977,Z 630.53,A -85,B 0,C 180,E1 -2056.524,E2 -2056.524} C_VEL
LIN {X 0,Y 572.945,Z 633.757,A -85,B 0,C 180,E1 -2057.964,E2 -2057.964} C_VEL
LIN {X 0,Y 572.981,Z 635.707,A -85,B 0,C 180,E1 -2059.399,E2 -2059.399} C_VEL
LIN {X 0,Y 572.92,Z 636.457,A -85,B 0,C 180,E1 -2060.824,E2 -2060.824} C_VEL
LIN {X 0,Y 572.975,Z 636.05,A -85,B 0,C 180,E1 -2062.246,E2 -2062.246} C_VEL
LIN {X 0,Y 572.974,Z 634.494,A -85,B 0,C 180,E1 -2063.663,E2 -2063.663} C_VEL
LIN {X 0,Y 572.942,Z 631.772,A -85,B 0,C 180,E1 -2065.075,E2 -2065.075} C_VEL
LIN {X 0,Y 573.049,Z 627.825,A -85,B 0,C 180,E1 -2066.485,E2 -2066.485} C_VEL
LIN {X 0,Y 572.995,Z 622.56,A -85,B 0,C 180,E1 -2067.892,E2 -2067.892} C_VEL
LIN {X 0,Y 573.11,Z 615.87,A -85,B 0,C 180,E1 -2069.298,E2 -2069.298} C_VEL
LIN {X 0,Y 573.206,Z 607.595,A -85,B 0,C 180,E1 -2070.703,E2 -2070.703} C_VEL
LIN {X 0,Y 573.293,Z 598.809,A -85,B 0,C 180,E1 -2071.932,E2 -2071.932} C_VEL
LIN {X 0,Y 573.446,Z 588.312,A -85,B 0,C 180,E1 -2073.162,E2 -2073.162} C_VEL
LIN {X 0,Y 573.625,Z 577.572,A -85,B 0,C 180,E1 -2074.216,E2 -2074.216} C_VEL
LIN {X 0,Y 573.784,Z 565.905,A -85,B 0,C 180,E1 -2075.183,E2 -2075.183} C_VEL
LIN {X 0,Y 573.999,Z 553.205,A -85,B 0,C 180,E1 -2076.062,E2 -2076.062} C_VEL
LIN {X 0,Y 574.213,Z 539.251,A -85,B 0,C 180,E1 -2076.854,E2 -2076.854} C_VEL
LIN {X 0,Y 574.382,Z 524.956,A -85,B 0,C 180,E1 -2077.501,E2 -2077.501} C_VEL
LIN {X 0,Y 574.555,Z 509.927,A -85,B 0,C 180,E1 -2078.02,E2 -2078.02} C_VEL
LIN {X 0,Y 574.666,Z 494.701,A -85,B 0,C 180,E1 -2078.395,E2 -2078.395} C_VEL
LIN {X 0,Y 574.747,Z 473.928,A -85,B 0,C 180,E1 -2078.704,E2 -2078.704} C_VEL
LIN {X 0,Y 575.01,Z 364.684,A -85,B 0,C 180,E1 -2080.103,E2 -2080.103} C_VEL
LIN {X 0,Y 573.212,Z 359.707,A -85,B 0,C 180,E1 -2080.241,E2 -2080.241} C_VEL
LIN {X 0,Y 573.222,Z 359.703,A -85,B 0,C 180,E1 -2082.03,E2 -2082.03} C_VEL
LIN {X 0,Y 573.211,Z 359.713,A -85,B 0,C 180,E1 -2084.92,E2 -2084.92} C_VEL
LIN {X 0,Y 573.199,Z 359.704,A -85,B 0,C 180,E1 -2087.85,E2 -2087.85} C_VEL
LIN {X 0,Y 573.195,Z 359.705,A -85,B 0,C 180,E1 -2090.078,E2 -2090.078} C_VEL
LIN {X 0,Y 573.184,Z 359.707,A -85,B 0,C 180,E1 -2092.34,E2 -2092.34} C_VEL
LIN {X 0,Y 573.189,Z 359.713,A -85,B 0,C 180,E1 -2094.86,E2 -2094.86} C_VEL
LIN {X 0,Y 573.186,Z 359.715,A -85,B 0,C 180,E1 -2096.979,E2 -2096.979} C_VEL
LIN {X 0,Y 573.193,Z 359.706,A -85,B 0,C 180,E1 -2099.478,E2 -2099.478} C_VEL
LIN {X 0,Y 573.219,Z 359.702,A -85,B 0,C 180,E1 -2102.222,E2 -2102.222} C_VEL
LIN {X 0,Y 573.211,Z 359.707,A -85,B 0,C 180,E1 -2104.767,E2 -2104.767} C_VEL
LIN {X 0,Y 573.213,Z 359.703,A -85,B 0,C 180,E1 -2107.809,E2 -2107.809} C_VEL
LIN {X 0,Y 573.206,Z 359.703,A -85,B 0,C 180,E1 -2110.527,E2 -2110.527} C_VEL
LIN {X 0,Y 573.188,Z 359.712,A -85,B 0,C 180,E1 -2113.363,E2 -2113.363} C_VEL
LIN {X 0,Y 573.196,Z 359.704,A -85,B 0,C 180,E1 -2116.335,E2 -2116.335} C_VEL
LIN {X 0,Y 573.24,Z 359.705,A -85,B 0,C 180,E1 -2119.474,E2 -2119.474} C_VEL
LIN {X 0,Y 573.182,Z 359.705,A -85,B 0,C 180,E1 -2122.188,E2 -2122.188} C_VEL
LIN {X 0,Y 573.214,Z 359.712,A -85,B 0,C 180,E1 -2125.23,E2 -2125.23} C_VEL
LIN {X 0,Y 573.208,Z 359.703,A -85,B 0,C 180,E1 -2128.182,E2 -2128.182} C_VEL
LIN {X 0,Y 573.216,Z 359.702,A -85,B 0,C 180,E1 -2130.631,E2 -2130.631} C_VEL
LIN {X 0,Y 573.181,Z 359.713,A -85,B 0,C 180,E1 -2133.516,E2 -2133.516} C_VEL
LIN {X 0,Y 573.185,Z 359.705,A -85,B 0,C 180,E1 -2136.132,E2 -2136.132} C_VEL
LIN {X 0,Y 573.235,Z 359.706,A -85,B 0,C 180,E1 -2139.173,E2 -2139.173} C_VEL
LIN {X 0,Y 573.188,Z 359.714,A -85,B 0,C 180,E1 -2141.41,E2 -2141.41} C_VEL
LIN {X 0,Y 573.208,Z 359.709,A -85,B 0,C 180,E1 -2143.62,E2 -2143.62} C_VEL
LIN {X 0,Y 573.226,Z 359.703,A -85,B 0,C 180,E1 -2145.806,E2 -2145.806} C_VEL
LIN {X 0,Y 573.252,Z 359.693,A -85,B 0,C 180,E1 -2148.745,E2 -2148.745} C_VEL
LIN {X 0,Y 573.221,Z 359.709,A -85,B 0,C 180,E1 -2151.539,E2 -2151.539} C_VEL
LIN {X 0,Y 573.207,Z 359.71,A -85,B 0,C 180,E1 -2153.664,E2 -2153.664} C_VEL
LIN {X 0,Y 573.185,Z 359.71,A -85,B 0,C 180,E1 -2155.781,E2 -2155.781} C_VEL
LIN {X 0,Y 573.274,Z 359.697,A -85,B 0,C 180,E1 -2157.892,E2 -2157.892} C_VEL
LIN {X 0,Y 573.285,Z 359.696,A -85,B 0,C 180,E1 -2160,E2 -2160} C_VEL
LIN {X 0,Y 573.264,Z 359.696,A -85,B 0,C 180,E1 -2162.811,E2 -2162.811} C_VEL
LIN {X 0,Y 573.256,Z 359.706,A -85,B 0,C 180,E1 -2165.628,E2 -2165.628} C_VEL
LIN {X 0,Y 573.211,Z 359.701,A -85,B 0,C 180,E1 -2168.46,E2 -2168.46} C_VEL
LIN {X 0,Y 573.26,Z 359.701,A -85,B 0,C 180,E1 -2171.312,E2 -2171.312} C_VEL
LIN {X 0,Y 573.224,Z 359.7,A -85,B 0,C 180,E1 -2174.406,E2 -2174.406} C_VEL
LIN {X 0,Y 573.18,Z 359.709,A -85,B 0,C 180,E1 -2177.114,E2 -2177.114} C_VEL
LIN {X 0,Y 573.192,Z 359.709,A -85,B 0,C 180,E1 -2180.079,E2 -2180.079} C_VEL
LIN {X 0,Y 573.184,Z 359.706,A -85,B 0,C 180,E1 -2182.34,E2 -2182.34} C_VEL
LIN {X 0,Y 573.219,Z 359.707,A -85,B 0,C 180,E1 -2185.412,E2 -2185.412} C_VEL
LIN {X 0,Y 573.183,Z 359.711,A -85,B 0,C 180,E1 -2188.018,E2 -2188.018} C_VEL
LIN {X 0,Y 573.207,Z 359.703,A -85,B 0,C 180,E1 -2190.88,E2 -2190.88} C_VEL
LIN {X 0,Y 573.232,Z 359.705,A -85,B 0,C 180,E1 -2193.521,E2 -2193.521} C_VEL
LIN {X 0,Y 573.175,Z 359.713,A -85,B 0,C 180,E1 -2196.054,E2 -2196.054} C_VEL
LIN {X 0,Y 573.206,Z 359.702,A -85,B 0,C 180,E1 -2198.704,E2 -2198.704} C_VEL
LIN {X 0,Y 573.19,Z 359.709,A -85,B 0,C 180,E1 -2201.46,E2 -2201.46} C_VEL
LIN {X 0,Y 573.197,Z 359.707,A -85,B 0,C 180,E1 -2204.337,E2 -2204.337} C_VEL
LIN {X 0,Y 573.212,Z 359.705,A -85,B 0,C 180,E1 -2207.362,E2 -2207.362} C_VEL
LIN {X 0,Y 573.225,Z 359.702,A -85,B 0,C 180,E1 -2210.571,E2 -2210.571} C_VEL
LIN {X 0,Y 573.208,Z 359.704,A -85,B 0,C 180,E1 -2213.075,E2 -2213.075} C_VEL
LIN {X 0,Y 573.239,Z 359.706,A -85,B 0,C 180,E1 -2215.67,E2 -2215.67} C_VEL
LIN {X 0,Y 573.214,Z 359.713,A -85,B 0,C 180,E1 -2218.183,E2 -2218.183} C_VEL
LIN {X 0,Y 573.242,Z 359.841,A -85,B 0,C 180,E1 -2219.43,E2 -2219.43} C_VEL
LIN {X 0,Y 575.476,Z 368.596,A -85,B 0,C 180,E1 -2220.375,E2 -2220.375} C_VEL
LIN {X 0,Y 575.45,Z 393.48,A -85,B 0,C 180,E1 -2222.743,E2 -2222.743} C_VEL
LIN {X 0,Y 574.95,Z 423.23,A -85,B 0,C 180,E1 -2225.635,E2 -2225.635} C_VEL
LIN {X 0,Y 574.532,Z 454.947,A -85,B 0,C 180,E1 -2228.659,E2 -2228.659} C_VEL
LIN {X 0,Y 574.307,Z 473.491,A -85,B 0,C 180,E1 -2230.383,E2 -2230.383} C_VEL
LIN {X 0,Y 575.176,Z 480.173,A -85,B 0,C 180,E1 -2230.5,E2 -2230.5} C_VEL
LIN {X 0,Y 574.761,Z 641.511,A -85,B 0,C 180,E1 -2232.589,E2 -2232.589} C_VEL
LIN {X 0,Y 574.626,Z 656.713,A -85,B 0,C 180,E1 -2232.931,E2 -2232.931} C_VEL
LIN {X 0,Y 574.44,Z 672.046,A -85,B 0,C 180,E1 -2233.428,E2 -2233.428} C_VEL
LIN {X 0,Y 574.291,Z 685.772,A -85,B 0,C 180,E1 -2234.017,E2 -2234.017} C_VEL
LIN {X 0,Y 574.048,Z 699.244,A -85,B 0,C 180,E1 -2234.739,E2 -2234.739} C_VEL
LIN {X 0,Y 573.86,Z 712.818,A -85,B 0,C 180,E1 -2235.632,E2 -2235.632} C_VEL
LIN {X 0,Y 573.635,Z 725.35,A -85,B 0,C 180,E1 -2236.629,E2 -2236.629} C_VEL
LIN {X 0,Y 573.477,Z 735.749,A -85,B 0,C 180,E1 -2237.616,E2 -2237.616} C_VEL
LIN {X 0,Y 573.286,Z 745.77,A -85,B 0,C 180,E1 -2238.734,E2 -2238.734} C_VEL
LIN {X 0,Y 573.243,Z 754.857,A -85,B 0,C 180,E1 -2239.938,E2 -2239.938} C_VEL
LIN {X 0,Y 573.133,Z 762.733,A -85,B 0,C 180,E1 -2241.183,E2 -2241.183} C_VEL
LIN {X 0,Y 573.075,Z 770.089,A -85,B 0,C 180,E1 -2242.601,E2 -2242.601} C_VEL
LIN {X 0,Y 573.04,Z 775.923,A -85,B 0,C 180,E1 -2244.016,E2 -2244.016} C_VEL
LIN {X 0,Y 572.951,Z 779.384,A -85,B 0,C 180,E1 -2245.074,E2 -2245.074} C_VEL
LIN {X 0,Y 573.004,Z 782.888,A -85,B 0,C 180,E1 -2246.484,E2 -2246.484} C_VEL
LIN {X 0,Y 572.935,Z 785.192,A -85,B 0,C 180,E1 -2247.891,E2 -2247.891} C_VEL
LIN {X 0,Y 572.938,Z 786.349,A -85,B 0,C 180,E1 -2249.297,E2 -2249.297} C_VEL
LIN {X 0,Y 572.938,Z 786.349,A -85,B 0,C 180,E1 -2250.703,E2 -2250.703} C_VEL
LIN {X 0,Y 572.935,Z 785.191,A -85,B 0,C 180,E1 -2252.109,E2 -2252.109} C_VEL
LIN {X 0,Y 573.004,Z 782.887,A -85,B 0,C 180,E1 -2253.516,E2 -2253.516} C_VEL
LIN {X 0,Y 572.951,Z 779.386,A -85,B 0,C 180,E1 -2254.925,E2 -2254.925} C_VEL
LIN {X 0,Y 573.012,Z 774.61,A -85,B 0,C 180,E1 -2256.337,E2 -2256.337} C_VEL
